# B&R Automation Studio project AS (part 3)

### paiHmiDropdwMenuRT.typ - Global data types
```iecst
(********************************************************************
 * COPYRIGHT -- pai
 ********************************************************************
 * Package: HMI
 * File: HMI.typ
 * Author: goran
 * Created: August 28, 2013
 ********************************************************************
 * Data types of package HMI
 ********************************************************************)
(*########################################################################*)
(*HMI object - Dropdown Menu located at the Upper Right side of the screen*)
(*########################################################################*)

TYPE
	paiHmiDropdwMenuRT_typ : 	STRUCT
		iMenuIndexRT : INT;
		iMenuRTTimeout : REAL; (*Duration after which a dropdown menu is automaticaly hiden if not clicked *)
		oMenuIndexRT : INT; (*Main menu currently selected menu item - RT*)
		oMenuVisible : INT;
		oMenuVisibleItems : ARRAY[0..paiHMI_ENUM_MENU_ITEMS_RT]OF INT; (*1-items is not visible*)
		oMenuDisabledItems : ARRAY[0..paiHMI_ENUM_MENU_ITEMS_RT]OF BOOL; (*1-Item is disabled*)
		iMenuSelectItem : ARRAY[0..paiHMI_ENUM_MENU_ITEMS_RT]OF BOOL; (*an input array to select items from the code; first found 1 will be selected;*)
		oMenuSelectedItems : ARRAY[0..paiHMI_ENUM_MENU_ITEMS_RT]OF BOOL; (*1-Item is currently selected (indexRT)*)
		oMenuPressedItems : ARRAY[0..paiHMI_ENUM_MENU_ITEMS_RT]OF BOOL; (*1-an item that was pressed, single shot*)
		mMenuVisibleOld : INT;
		menuRTHideTimer : TON;
	END_STRUCT;
END_TYPE
```

### paiHmiAlert.h
```c
/********************************************************************
 * COPYRIGHT -- pai
 ********************************************************************
 * Program: hmilogic
 * File: hmiAlert.h
 * Author: goran
 * Created: September 05, 2013
 *******************************************************************/

#include <bur/plctypes.h>
#ifdef _DEFAULT_INCLUDES
#include <AsDefault.h>
#endif
void paiHmiAlertHide(paiHmiAlert_typ* p);
BOOL paiHmiAlertIsActive(paiHmiAlert_typ* p);
void paiHmiAlertShow(paiHmiAlert_typ* p, char* headerText, char* alertText, UDINT alertDuration);
void paiHmiAlertCyclic(paiHmiAlert_typ* p);
```

### paiHmiSystemDateTime.c
```c
/********************************************************************
 * COPYRIGHT -- pai
 ********************************************************************
 * Program: hmilogic
 * File: hmiAlert.c
 * Author: goran
 * Created: September 05, 2013
 *******************************************************************/

#include <bur/plctypes.h>
#ifdef _DEFAULT_INCLUDES
	#include <AsDefault.h>
#endif

void paiHmiSystemDateTimeInit(paiHmiSystemTime_typ* p)
{
}
void paiHmiSystemDateTimeCyclic(paiHmiSystemTime_typ* p)
{
	if(!p->iChangeTimeRequest){
		p->mGetTime.enable = 1;
		p->mGetTime.DT1 = (UDINT)&p->mDateTime;
		DTGetTime(&p->mGetTime);
		p->mDateTime = p->mGetTime.DT1;
		DT_TO_DTStructure(p->mDateTime, (UDINT)&p->oDateTimeActual);
	}else{
		p->iChangeTimeRequest = 0;
		p->mDateTime = DTStructure_TO_DT((UDINT)&p->oDateTimeActual);
		p->mSetTime.enable = 1;
		p->mSetTime.DT1 = p->mDateTime;
		DTSetTime(&p->mSetTime);
	}

}
//eof
```

### paiHmiParamList.h
```c
/********************************************************************
 * COPYRIGHT -- pai
 ********************************************************************
 * Program: hmilogic
 * File: hmiParamList.h
 * Author: goran
 * Created: September 05, 2013
 *******************************************************************/
#include <bur/plctypes.h>
#ifdef _DEFAULT_INCLUDES
#include <AsDefault.h>
#endif
//void hmiParamListTableCyclic(hmiParamListTable_typ* p);
void hmiParamListTableEntryLast(hmiParamListTable_typ* p);
void hmiParamListTableEntryFirst(hmiParamListTable_typ* p, char* pListName);
 void hmiParamListTableAddEntryNext(hmiParamListTable_typ* p, UDINT pValue, char* pName, REAL valDefault, REAL valMin, REAL valMax, int decPlaces, REAL k_factor, REAL n_factor, UINT valueType, char* pDescription);
```

### paiHMI.var
```iecst
(********************************************************************
 * COPYRIGHT -- pai
 ********************************************************************
 * Package: HMI
 * File: HMI.var
 * Author: goran
 * Created: August 28, 2013
 ********************************************************************
 * Variables of package HMI
 ********************************************************************)
VAR
	gPaiHmiMain : paiHmiTemplate_typ; (*HMI logic, page navigation, visibility control, etc.*)
	gPaiHmiMsgScroll : paiHmiMsgScrolling_typ; (*Scrolling Alarm Msg Support*)
	gPaiHmiDialogMsg : paiHmiDialog_typ; (*Scrolling Alarm Msg Support*)
	gPaiHmiAlertMsg : paiHmiAlert_typ; (*Scrolling Alarm Msg Support*)
	gPaiHmiRTMenu : paiHmiDropdwMenuRT_typ;
	gPaiHmiSystemDateTime : paiHmiSystemTime_typ;
	gPaiHmiNetworking : paiHmiSystemNetworking_typ;
END_VAR
VAR RETAIN
	gScrensaverTimeout : INT := 0;
END_VAR
```

### Program Logical/paiComponents/paiTemplate/paiHMI/paiHmi (ANSIC)

- paiHmiSystemDateTime.c (reference to Logical/paiComponents/paiHmi/paiHmiSystemDateTime.c)

### cfgUdpApp.typ - Package data types
```iecst
(********************************************************************
 * COPYRIGHT --
 ********************************************************************
 * Package: UDP
 * File: cfgUdpApp.typ
 * Author: goran
 * Created: October 15, 2014
 ********************************************************************
 * Data types of package UDP
 ********************************************************************)

TYPE
	cfgUdpApp_typ : 	STRUCT
		test1 : UDINT;
		test2 : UDINT;
	END_STRUCT;
END_TYPE
```

- Program Logical/paiComponents/paiUser/paiUser (ANSIC) (no source held here)

### Safety_var.var
```iecst
(*Global PV containing the safety variables.*)
VAR RETAIN
	gSafetyPermInfo : paiSL_Perm_Info_typ;
END_VAR
(*Insert your comment here.*)
VAR
	gSafety : paiSL_typ;
END_VAR
(*Defined constants- change based on specific commissioning configuration*)
VAR
	DEFINE_OFFSET_ERR_START : UDINT := 100000;
END_VAR
VAR CONSTANT
	DEFINE_SAFETY_APP_ID : UINT := 1;
	DEFINE_TIME_MAX_RCTRL_CMD : REAL := 30;
	DEFINE_TIME_ERROR_AUTORESET : REAL := 5;
	DEFINE_TIME_SCANNING_RETRY : REAL := 10;
	DEFINE_TIME_PRINT_HMI_STATUS : REAL := 2;
	DEFINE_SAFELOGIC_ADDRESS : STRING[80] := 'SL1.IF1.ST4.IF1.ST2';
	DEFINE_VERSION : UINT := safeVERSION_R107;
	DEFINE_SAFELOGIC_ID : UINT := 1;
END_VAR
```

### Program Logical/pkgSafety/SafeINIT (IEC)

#### Action_Reset_FBK.st
```iecst
ACTION Action_Reset_FBK:
	gSafety.prv.FBK.RemoteControl.Execute := FALSE;
	gSafety.prv.FBK.DownloadApplication.Execute := FALSE;
	gSafety.prv.FBK.UDID_High.enable := FALSE;
	gSafety.prv.FBK.UDID_Low.enable := FALSE;
END_ACTION
```

### Data object Logical/acp10etxen (Ett)

- acp10etxen.ett (not shown)

- Project.language (not shown)

### Package Logical/HMI - HMI screens 

- Visualisation Logical/HMI/WSVGA (not shown)

### HMImsgScroll.typ - not listed in the package file held
```iecst
(********************************************************************
 * COPYRIGHT -- piedmont
 ********************************************************************
 * Package: HMI
 * File: HMI.typ
 * Author: goran
 * Created: August 28, 2013
 ********************************************************************
 * Data types of package HMI
 ********************************************************************)
(*########################################################################*)
(*HMI object - Scrolling Messages (i.e. alarms)*)
(*########################################################################*)

TYPE
	hmiMsgScrolling_typ : 	STRUCT
		iAdrAlarmArray : UDINT; (*input: address of the alarm array*)
		iAlarmArrayLen : UDINT; (*input: number of alarms in the alarm array*)
		iMsgTimeXms : UDINT; (*input: duration of the message display (if more than one message/alarm active)*)
		oMsgID : UINT; (*output: message ID of the active alarm / message*)
		oMsgVisible : UINT; (*output: visibilty control DP for the VC text message*)
		state : UINT; (*Status for common dialog layer*)
		tmr1 : TON; (*Dialog control timer*)
	END_STRUCT;
END_TYPE
```

### Program Logical/HMI/hmilogic

#### hmiAlert.c
```c
/********************************************************************
 * COPYRIGHT -- piedmont
 ********************************************************************
 * Program: hmilogic
 * File: hmiAlert.c
 * Author: goran
 * Created: September 05, 2013
 *******************************************************************/

#include <bur/plctypes.h>
#ifdef _DEFAULT_INCLUDES
	#include <AsDefault.h>
#endif

/**
Bit manipulaiton utility functions.
 */
//#include <../../bglib/bgBitUtilities.h>

/**
String manipulaiton utility functions.
 */
//#include <../../bglib/bgsprintf.h>
//#include <../../bglib/bgstring.h>

/**
 Timer control utility functions.
 */
//#include <../../bglib/bgTimer1ms.h>

//Control on/off a variable that control the visibility of the alarm alert display
void hmiAlertHide(hmiAlert_typ* p)
{
	//control visibility of the layer > make it invisible
	bgBitSetUINT(&p->status, 0, 1);
}

// Is alert message active (visible)?
BOOL hmiAlertIsActive(hmiAlert_typ* p)
{
	if(bgTimerIsTimeOut(&p->tmr1))
		return 0;
	else
		return 1;
}

// Show the alert with a specified text and for a selected amount of time
void hmiAlertShow(hmiAlert_typ* p, char* alertText, UDINT alertDuration)
{
	//control visibility of the layer > make it visible
	bgBitSetUINT(&p->status, 0, 0);
	bgStrCpyN(p->message, alertText, sizeof(p->message));
	bgTimerStart(&p->tmr1, alertDuration);
}

// Cyclic operation of the alert box.
void hmiAlertCyclic(hmiAlert_typ* p)
{
	bgTimerCyclic(&p->tmr1);
	if( !(p->status & 0x1) && bgTimerIsTimeOut(&p->tmr1) ){
		hmiAlertHide(p);
	}
}
//eof
```

#### hmiDialog.c
```c
/********************************************************************
 * COPYRIGHT -- piedmont
 ********************************************************************
 * Program: hmilogic
 * File: hmiDialog.c
 * Author: goran
 * Created: September 05, 2013
 *******************************************************************/

#include <bur/plctypes.h>
#ifdef _DEFAULT_INCLUDES
	#include <AsDefault.h>
#endif

/*
###############################################################################
Simple dialog support w. OK and Cancle response
###############################################################################
*/

/**
Find if HMI dialog is active (visible) or not
\param p prt to hmiDialog_typ structure
\return 0 not active (not visible)
\return 1 active (visible)
*/
BOOL hmiDialogIsActive(hmiDialog_typ* p)
{
	//hide the dialog
	if(p->status & 0x1){
		return 0; //not visible > not active
	}

	return 1; //visible > active
}

/**
Hide HMI dialog (make it not visible)
\param p prt to hmiDialog_typ structure
*/
void hmiDialogHide(hmiDialog_typ* p)
{
	//hide the dialog
	bgBitSetUINT(&p->status, 0, 1);

	//define the message
	strcpy(p->message, "");
}

/**
Hide HMI dialog (make it not visible)
\param p prt to hmiDialog_typ structure
\param msg text message that will be displayed in a dialog
\param timeout_ms time duration to show the dialog. Upon timer expiration, dialog will automatically generate either ok or cancel (configured, see timeoutConfig)
\param resultForOk value returned in case user response is OK (if 0, default is used = 1)
\param resultForCancel value returned in case user response is Cancel ((if 0, default is used = 2)
\param timeoutConfig 0-timeout wil return value for Cancel, 1-timeout will return value for OK
*/
 void hmiDialogShow(hmiDialog_typ* p, char* msg, UINT timeout_ms, UINT resultForOk, UINT resultForCancel, UINT timeoutConfig)
{
	//show the dialog
	bgBitSetUINT(&p->status, 0, 0);

	//define the message
	bgStrCpyN(p->message, msg, sizeof(p->message));

	//start the timer
	bgTimerStart(&p->tmr1, timeout_ms);

	//set the result to 0 (not complete)
	p->result = 0;
	p->btnOk = 0;
	p->btnCancel = 0;

	//configuration of the timeout
	p->timeoutConfig = timeoutConfig;

	p->resultForOk = resultForOk;
	if(!p->resultForOk)
		p->resultForOk = 1;

	p->resultForCancel = resultForCancel;
	if(!p->resultForCancel)
		p->resultForCancel = 2;

}

/**
Hide HMI dialog cyclic routine
\param p prt to hmiDialog_typ structure
*/
UINT hmiDialogCyclic(hmiDialog_typ* p)
{
	//operate timer always
	bgTimerCyclic(&p->tmr1);

	p->tmr1RemainingTimeSec = (p->tmr1.PT - p->tmr1.ET) / 1000;

	//if dialog not visible > nothing to do
	if(p->status)
		return 0;

	if( bgTimerIsTimeOut(&p->tmr1) ){
		//hide the dialog
		hmiDialogHide(p);
		//check how is the timeout configured and generate such result
		if(!p->timeoutConfig){
			p->result = p->resultForCancel;
			return p->resultForCancel; //return cancel
		}
		p->result = p->resultForOk;
		return p->resultForOk;//return OK
	}

	//keep checking if OK or Cancel buttons are pressed
	if( p->btnOk || p->btnCancel ){

		//hide the dialog
		hmiDialogHide(p);

		//return user's selection:
		if(p->btnOk){
			p->result = p->resultForOk;
		}else
		if(p->btnCancel){
			p->result = p->resultForCancel;
		}

		p->btnOk = 0;
		p->btnCancel = 0;

		return p->result; //return user's selection
	}
	return 0; //no button pressed
}
//EOF
```

### ParStructs.typ
```iecst
(*Insert your comment here.*)

TYPE
	Global_Rec_Cfg_typ : 	STRUCT
		Rec : Global_Rec_typ;
		Cfg : Global_Cfg_typ;
	END_STRUCT;
END_TYPE

(*Insert your comment here.*)

TYPE
	Global_RecCfg_Public_In_typ : 	STRUCT
		Copy_save_to_active : USINT;
		Copy_active_to_save : USINT;
		FileName : STRING[255];
	END_STRUCT;
	Global_RecCfg_Public_Out_typ : 	STRUCT
		save_differs_from_active : USINT;
	END_STRUCT;
	Global_Rec_Cfg_Info_typ : 	STRUCT
		O : Global_RecCfg_Public_Out_typ;
		I : Global_RecCfg_Public_In_typ;
	END_STRUCT;
	Global_Rec_Cfg_IO_typ : 	STRUCT
		Rec : Global_Rec_Cfg_Info_typ;
		Cfg : Global_Rec_Cfg_Info_typ;
	END_STRUCT;
END_TYPE

(*Insert your comment here.*)

TYPE
	Global_Par_typ : 	STRUCT
		save : Global_Rec_Cfg_typ;
		active : Global_Rec_Cfg_typ;
		IO : Global_Rec_Cfg_IO_typ;
	END_STRUCT;
END_TYPE
```

### RecCfg.var
```iecst
VAR CONSTANT
	DEFINE_CONSTANT_MAGIC_PREFIX : UDINT := 16#12345678;
	DEFINE_CONSTANT_MAGIC_SUFFIX : UDINT := 16#87654321;
END_VAR
(*Insert your comment here.*)
VAR CONSTANT
	MAX_IDX_TOTAL_RECIPES : UINT := 100;
END_VAR
(*Insert your comment here.*)
VAR RETAIN
	gConfigName : STRING[255];
	gRecipeName : STRING[255];
END_VAR
(*Insert your comment here.*)
VAR RETAIN
	gRecCfg : Global_Par_typ;
END_VAR
```

### Program Logical/pkgRecCfg/Recipe_Handling (IEC)

#### Init.st - Init code
```iecst
PROGRAM _INIT
	IF gRecCfg.active.Cfg.MagicPrefix <> DEFINE_CONSTANT_MAGIC_PREFIX OR gRecCfg.save.Cfg.MagicPrefix <> DEFINE_CONSTANT_MAGIC_PREFIX
		OR gRecCfg.active.Cfg.MagicSuffix <> DEFINE_CONSTANT_MAGIC_SUFFIX OR gRecCfg.save.Cfg.MagicSuffix <> DEFINE_CONSTANT_MAGIC_SUFFIX THEN

		brsmemset(ADR(gRecCfg.save.Cfg), 0, SIZEOF(Global_Cfg_typ));
		brsmemset(ADR(gRecCfg.active.Cfg), 0, SIZEOF(Global_Cfg_typ));

		gRecCfg.active.Cfg.MagicPrefix := DEFINE_CONSTANT_MAGIC_PREFIX;
		gRecCfg.save.Cfg.MagicPrefix:= DEFINE_CONSTANT_MAGIC_PREFIX;

		gRecCfg.active.Cfg.MagicSuffix := DEFINE_CONSTANT_MAGIC_SUFFIX;
		gRecCfg.save.Cfg.MagicSuffix:= DEFINE_CONSTANT_MAGIC_SUFFIX;
		//
//		brsmemset(ADR(gLinePermData), 0, SIZEOF(Line_Permanent_Variables_typ));
//		brsmemset(ADR(gStatistics), 0, SIZEOF(Global_Statistics_typ));
//		brsmemset(ADR(Axis_Line_Par), 0, SIZEOF(MpAxisBasicParType));
//		brsmemset(ADR(Axis_Blank_Par), 0, SIZEOF(MpAxisBasicParType));
//		brsmemset(ADR(Axis_Coupling_Master_Line_Par), 0, SIZEOF(MpAxisCouplingParType));
//
//		Set_Default_Config_Values(pCfg := ADR(gRecCfg.defaultvals.Cfg), MachineType := gMachineType);
//		Set_Default_Config_Values(pCfg := ADR(gRecCfg.save.Cfg), MachineType := gMachineType);
//		Set_Default_Config_Values(pCfg := ADR(gRecCfg.active.Cfg), MachineType := gMachineType);
//
//		gRecipeName := 'No Config';
//
//		gAlarms.RecCfg.Default_Cfg_Set := TRUE;

//		SYSreset(1, 1);
	END_IF;

	IF gRecCfg.active.Rec.MagicPrefix <> DEFINE_CONSTANT_MAGIC_PREFIX OR gRecCfg.save.Rec.MagicPrefix <> DEFINE_CONSTANT_MAGIC_PREFIX
		OR gRecCfg.active.Rec.MagicSuffix <> DEFINE_CONSTANT_MAGIC_SUFFIX OR gRecCfg.save.Rec.MagicSuffix <> DEFINE_CONSTANT_MAGIC_SUFFIX THEN

		brsmemset(ADR(gRecCfg.save.Rec), 0, SIZEOF(Global_Rec_typ));
		brsmemset(ADR(gRecCfg.active.Rec), 0, SIZEOF(Global_Rec_typ));

		gRecCfg.active.Rec.MagicPrefix := DEFINE_CONSTANT_MAGIC_PREFIX;
		gRecCfg.save.Rec.MagicPrefix:= DEFINE_CONSTANT_MAGIC_PREFIX;

		gRecCfg.active.Rec.MagicSuffix := DEFINE_CONSTANT_MAGIC_SUFFIX;
		gRecCfg.save.Rec.MagicSuffix:= DEFINE_CONSTANT_MAGIC_SUFFIX;
		//
//		brsmemset(ADR(gLinePermData), 0, SIZEOF(Line_Permanent_Variables_typ));
//		brsmemset(ADR(gStatistics), 0, SIZEOF(Global_Statistics_typ));
//		brsmemset(ADR(Axis_Line_Par), 0, SIZEOF(MpAxisBasicParType));
//		brsmemset(ADR(Axis_Blank_Par), 0, SIZEOF(MpAxisBasicParType));
//		brsmemset(ADR(Axis_Coupling_Master_Line_Par), 0, SIZEOF(MpAxisCouplingParType));
//
//		Set_Default_Recipe_Values(pRec := ADR(gRecCfg.defaultvals.Rec), MachineType := gMachineType);
//		Set_Default_Recipe_Values(pRec := ADR(gRecCfg.save.Rec), MachineType := gMachineType);
//		Set_Default_Recipe_Values(pRec := ADR(gRecCfg.active.Rec), MachineType := gMachineType);
//
//		gRecipeName := 'No Recipe';
//
//		gAlarms.RecCfg.Default_Rec_Set := TRUE;
//		SYSreset(1, 1);
	END_IF;

	gRecCfg.IO.Rec.I.FileName := 'rec1';
	gRecCfg.IO.Cfg.I.FileName := 'cfg1';

	Recipe_CSV_Control.MpLink := ADR(Recipe_CSV_MpLink);
	Recipe_CSV_Control.Enable := TRUE;
	Recipe_CSV_Control.DeviceName := ADR('Recipe');
	Recipe_CSV_Control.FileName := ADR(gRecCfg.IO.Rec.I.FileName);
	Recipe_CSV_Control.Category := ADR('Recipe');
	Recipe_CSV_Control.Header := ADR(Recipe_CSV_Header);

	Config_CSV_Control.MpLink := ADR(Config_CSV_MpLink);
	Config_CSV_Control.Enable := TRUE;
	Config_CSV_Control.DeviceName := ADR('Config');
	Config_CSV_Control.FileName := ADR(gRecCfg.IO.Cfg.I.FileName);
	Config_CSV_Control.Category := ADR('Config');
	Config_CSV_Control.Header := ADR(Config_CSV_Header);

	Recipe_CSV_RegPar.MpLink := ADR(Recipe_CSV_MpLink);
	Recipe_CSV_RegPar.Enable := TRUE;
	Recipe_CSV_RegPar.PVName := ADR('gRecCfg.save.Rec');
	Recipe_CSV_RegPar.Category := ADR('Recipe');

	Config_CSV_RegPar.MpLink := ADR(Config_CSV_MpLink);
	Config_CSV_RegPar.Enable := TRUE;
	Config_CSV_RegPar.PVName := ADR('gRecCfg.save.Cfg');
	Config_CSV_RegPar.Category := ADR('Config');

	Recipe_CSV_UI.MpLink := ADR(Recipe_CSV_MpLink);
	Recipe_CSV_UI.Enable := TRUE;
	Recipe_CSV_UI.UIConnect := ADR(gRecipe_CSV_UIConnect);

	Config_CSV_UI.MpLink := ADR(Config_CSV_MpLink);
	Config_CSV_UI.Enable := TRUE;
	Config_CSV_UI.UIConnect := ADR(gConfig_CSV_UIConnect);

	Recipe_CSV_UI.UISetup.RecipeListSize := 20;
	Recipe_CSV_UI.UISetup.RecipeListScrollWindow := 1;
	Recipe_CSV_UI.UISetup.Confirmation.RecipeCreate := TRUE;
	Recipe_CSV_UI.UISetup.Confirmation.RecipeLoad := TRUE;
	Recipe_CSV_UI.UISetup.Confirmation.RecipeSave := TRUE;
	Recipe_CSV_UI.UISetup.Confirmation.RecipeDelete := TRUE;

	Config_CSV_UI.UISetup.RecipeListSize := 20;
	Config_CSV_UI.UISetup.RecipeListScrollWindow := 1;
	Config_CSV_UI.UISetup.Confirmation.RecipeCreate := TRUE;
	Config_CSV_UI.UISetup.Confirmation.RecipeLoad := TRUE;
	Config_CSV_UI.UISetup.Confirmation.RecipeSave := TRUE;
	Config_CSV_UI.UISetup.Confirmation.RecipeDelete := TRUE;

	pRecCfgUIConnect ACCESS ADR(gRecipe_CSV_UIConnect);
	pCmd ACCESS ADR(loc.Rec.HMI);

	gRecipe_CSV_UIConnect.New.FileName := 'Rec_Name';
	gConfig_CSV_UIConnect.New.FileName := 'Cfg_Name';

	Recipe_CSV_Control;
	Recipe_CSV_RegPar;
	Recipe_CSV_UI;

	Config_CSV_Control;
	Config_CSV_RegPar;
	Config_CSV_UI;

END_PROGRAM
```

### Alarm.var
```iecst
VAR
	AlarmX_HistoryUI : MpAlarmXHistoryUI;
	AlarmX_History_UIConnect : MpAlarmXHistoryUIConnectType;
	AlarmX_ListUI : MpAlarmXListUI;
	AlarmX_ListUIConnect : MpAlarmXListUIConnectType;
	AlarmX_History : MpAlarmXHistory;
	AlarmX_Control : MpAlarmXCore;
END_VAR
(*Insert your comment here.*)
VAR
	Com_Logger_UI : MpComLoggerUI := (0);
	Com_Logger_UIConnect : MpComLoggerUIConnectType := (0);
END_VAR
```

### Program Logical/pkgAlert/AlarmX (IEC)

#### Types.typ
```iecst
TYPE
	MachineAlarm_typ : 	STRUCT
		str : {REDUND_UNREPLICABLE} STRING[80];
		active : {REDUND_UNREPLICABLE} BOOL;
	END_STRUCT;
	MachineReaction_typ : 	STRUCT
		str : {REDUND_UNREPLICABLE} STRING[80];
		active : {REDUND_UNREPLICABLE} BOOL;
	END_STRUCT;
	AlarmX_Local_TmpVar_typ : 	STRUCT
		val_float : {REDUND_UNREPLICABLE} REAL;
		ExampleAlarm : {REDUND_UNREPLICABLE} MachineAlarm_typ;
		ExampleReaction : {REDUND_UNREPLICABLE} MachineReaction_typ;
	END_STRUCT;
END_TYPE
```

### UserXVar.var
```iecst
VAR
	UserX_ManagerUI : MpUserXManagerUI;
	UserX_LoginUI : MpUserXLoginUI;
	UserX_Login : MpUserXLogin;
END_VAR
```

### Program Logical/pkgData/DataTask (IEC)

#### LocalFunctions.fun
```iecst
FUNCTION Register_Log_PV : BOOL (* *) (*$GROUP=User,$CAT=User,$GROUPICON=User.png,$CATICON=User.png*)
	VAR_INPUT
		pDesc : REFERENCE TO STRING[80]; (*pRegParBlock : REFERENCE TO MpDataRegPar;*)
		pPVName : REFERENCE TO STRING[80];
		pIterator : REFERENCE TO DINT;
		pMpLink : REFERENCE TO MpComIdentType;
	END_VAR
END_FUNCTION
```

#### Register_Log_PV.st
```iecst
FUNCTION Register_Log_PV

//	pRegParBlock.MpLink := ADR(pMpLink);
//	pRegParBlock.Enable := TRUE;
//	pRegParBlock.PVName := ADR(pPVName);
//	pRegParBlock.Description := ADR(pDesc);
//	pRegParBlock();

	pIterator := pIterator + 1;
	RETURN;
END_FUNCTION
```

### Program Logical/pkgData/File_Handling (IEC)

#### Init.st - Init code
```iecst
PROGRAM _INIT
	File_Manager_Control.MpLink := ADR(File_Manager_MpLink);
	File_Manager_Control.Enable := TRUE;
	File_Manager_Control.UIConnect := ADR(File_Manager_UIConnect);

	File_Manager_UIConnect.DeviceList.DeviceNames[0] := 'ROOT';
	File_Manager_UIConnect.DeviceList.DeviceNames[1] := 'Config';
	File_Manager_UIConnect.DeviceList.DeviceNames[2] := 'Recipe';
	File_Manager_UIConnect.DeviceList.DeviceNames[3] := 'Data_Log';
	File_Manager_UIConnect.DeviceList.DeviceNames[4] := 'USB1';
	File_Manager_UIConnect.DeviceList.DeviceNames[5] := 'USB2';

	File_Manager_Control.UISetup.FileListSize := 8;
	File_Manager_Control.UISetup.FileListScrollWindow := 5;

	File_Manager_Control;

END_PROGRAM
```

### Library Logical/pkgPVListView/paiPVTable (ANSIC)
Depends on: standard, sys_lib, wbrLogSvc, ArTextSys, bglibasWBR, jgLibC, Acp10par

#### Languages.typ
```iecst
TYPE
	Language_Enums :
		(
		LANGUAGE_ENGLISH := 0,
		LANGUAGE_SWEDISH := 1,
		LANGUAGE_PORTUGESE := 2,
		LANGUAGE_GERMAN := 3,
		LANGUAGE_FRENCH := 4,
		LANGUAGE_SPANISH := 5
		);
	Enum_PV_types :
		(
		PV_REAL,
		PV_UDINT
		);
END_TYPE
```

### Program Logical/pkgPVListView/HMITableManager (IEC)

#### Types.typ
```iecst
TYPE
	hmiTableRecCfgTrigger_typ : 	STRUCT
		Dispense : BOOL := FALSE;
		Inspect : BOOL := FALSE;
	END_STRUCT;
	hmiTableTrigger_typ : 	STRUCT
		Rec : hmiTableRecCfgTrigger_typ;
		Cfg : hmiTableRecCfgTrigger_typ;
	END_STRUCT;
	hmiTableLoad_typ : 	STRUCT
		Trigger : BOOL;
	END_STRUCT;
	hmiTables_typ : 	STRUCT
		Trigger : hmiTableTrigger_typ;
		Load : hmiTableLoad_typ;
	END_STRUCT;
	HMITableControlLocal_typ : 	STRUCT
		tables : hmiTables_typ;
	END_STRUCT;
END_TYPE
```

#### Main.st
```iecst
PROGRAM _INIT
	Init_Logbook.Enable := TRUE;
	Init_Logbook.Name := 'usr_table';
	Init_Logbook();

END_PROGRAM

//TODO: Load param array with %s, replace with index.
//TODO: More scrutiny to ensure tables were done correctly

PROGRAM _CYCLIC
	svnRevision;

//	IF loc.tables.Trigger.Rec.Dispense THEN
//		loc.tables.Trigger.Rec.Dispense := FALSE;
//		ActivateHMITable(gRecCfg.active.Cfg.HMI.MachineLang, pHMITable := ADR(gHmiParamTable), pTableValues := ADR(loadHMITable[TABLE_REC_DISPENSE].hmiStruct));
//	END_IF;
//
//	IF loc.tables.Trigger.Rec.Inspect THEN
//		loc.tables.Trigger.Rec.Inspect := FALSE;
//		ActivateHMITable(gRecCfg.active.Cfg.HMI.MachineLang, pHMITable := ADR(gHmiParamTable), pTableValues := ADR(loadHMITable[TABLE_REC_INSPECT].hmiStruct));
//	END_IF;
//
//	IF loc.tables.Trigger.Rec.Eject THEN
//		loc.tables.Trigger.Rec.Eject := FALSE;
//		ActivateHMITable(gRecCfg.active.Cfg.HMI.MachineLang, pHMITable := ADR(gHmiParamTable), pTableValues := ADR(loadHMITable[TABLE_REC_EJECT].hmiStruct));
//	END_IF;
//
//	IF loc.tables.Trigger.Rec.Motor THEN
//		loc.tables.Trigger.Rec.Motor := FALSE;
//		ActivateHMITable(gRecCfg.active.Cfg.HMI.MachineLang, pHMITable := ADR(gHmiParamTable), pTableValues := ADR(loadHMITable[TABLE_REC_MOTOR].hmiStruct));
//	END_IF;
//
//	IF loc.tables.Trigger.Rec.Process THEN
//		loc.tables.Trigger.Rec.Process := FALSE;
//		ActivateHMITable(gRecCfg.active.Cfg.HMI.MachineLang, pHMITable := ADR(gHmiParamTable), pTableValues := ADR(loadHMITable[TABLE_REC_PROCESS].hmiStruct));
//	END_IF;
//
//	IF loc.tables.Trigger.Rec.Loader THEN
//		loc.tables.Trigger.Rec.Loader := FALSE;
//		ActivateHMITable(gRecCfg.active.Cfg.HMI.MachineLang, pHMITable := ADR(gHmiParamTable), pTableValues := ADR(loadHMITable[TABLE_REC_LOADER].hmiStruct));
//	END_IF;
//
//	IF loc.tables.Trigger.Cfg.Dispense THEN
//		loc.tables.Trigger.Cfg.Dispense := FALSE;
//		ActivateHMITable(gRecCfg.active.Cfg.HMI.MachineLang, pHMITable := ADR(gHmiParamTable), pTableValues := ADR(loadHMITable[TABLE_CFG_DISPENSE].hmiStruct));
//	END_IF;
//
//	IF loc.tables.Trigger.Cfg.Inspect THEN
//		loc.tables.Trigger.Cfg.Inspect := FALSE;
//		ActivateHMITable(gRecCfg.active.Cfg.HMI.MachineLang, pHMITable := ADR(gHmiParamTable), pTableValues := ADR(loadHMITable[TABLE_CFG_INSPECT].hmiStruct));
//	END_IF;
//
//	IF loc.tables.Trigger.Cfg.Eject THEN
//		loc.tables.Trigger.Cfg.Eject := FALSE;
//		ActivateHMITable(gRecCfg.active.Cfg.HMI.MachineLang, pHMITable := ADR(gHmiParamTable), pTableValues := ADR(loadHMITable[TABLE_CFG_EJECT].hmiStruct));
//	END_IF;
//
//	IF loc.tables.Trigger.Cfg.Motor THEN
//		loc.tables.Trigger.Cfg.Motor := FALSE;
//		ActivateHMITable(gRecCfg.active.Cfg.HMI.MachineLang, pHMITable := ADR(gHmiParamTable), pTableValues := ADR(loadHMITable[TABLE_CFG_MOTOR].hmiStruct));
//	END_IF;
//
//	IF loc.tables.Trigger.Cfg.Process THEN
//		loc.tables.Trigger.Cfg.Process := FALSE;
//		ActivateHMITable(gRecCfg.active.Cfg.HMI.MachineLang, pHMITable := ADR(gHmiParamTable), pTableValues := ADR(loadHMITable[TABLE_CFG_PROCESS].hmiStruct));
//	END_IF;
//
//	IF loc.tables.Trigger.Cfg.Loader THEN
//		loc.tables.Trigger.Cfg.Loader := FALSE;
//		ActivateHMITable(gRecCfg.active.Cfg.HMI.MachineLang, pHMITable := ADR(gHmiParamTable), pTableValues := ADR(loadHMITable[TABLE_CFG_LOADER].hmiStruct));
//	END_IF;
//
//	IF loc.tables.Trigger.Cfg.Admin THEN
//		loc.tables.Trigger.Cfg.Admin := FALSE;
//		ActivateHMITable(gRecCfg.active.Cfg.HMI.MachineLang, pHMITable := ADR(gHmiParamTable), pTableValues := ADR(loadHMITable[TABLE_CFG_ADMIN].hmiStruct));
//	END_IF;
//
//	IF loc.tables.Load.Trigger THEN
//		SYSreset(1,1);
//	END_IF;
//
//	hmiParamListTableCyclic(ADR(gHmiParamTable));

END_PROGRAM

PROGRAM _EXIT
	(* Insert code here *)

END_PROGRAM
```

### Audit_Global.var
```iecst
VAR
	Audit_Control : MpAuditTrail := (0);
	Audit_Config : MpAuditTrailConfig := (0);
	Audit_Config_Struct : MpAuditTrailConfigType := (0);
	Audit_UI : MpAuditTrailUI := (0);
	Audit_UIConnect : MpAuditTrailUIConnectType := (0);
	Audit_VC4_Event : MpAuditVC4Event := (0);
END_VAR
```

### EnMon_Global.var
```iecst
VAR
	Energy_Control : MpEnergyCore;
	Energy_UI : MpEnergyCoreUI := (UISetup:=(ModuleListSize:=6));
	Energy_UIConnect : MpEnergyCoreUIConnectType;
END_VAR
```

### Program Logical/pkgEnMon/EnMon (IEC)

#### Main.st
```iecst
PROGRAM _INIT
	Energy_Control.MpLink := ADR(Energy_MpLink);
	Energy_Control.Enable := TRUE;
	Energy_Control.DeviceName := ADR('Energy');
	Energy_Control();
	Energy_UI.MpLink := ADR(Energy_MpLink);
	Energy_UI.Enable := TRUE;
	Energy_UI.UISetup.ModuleListSize := 5;
	Energy_UI.UISetup.ModuleScrollWindow := 10;
	Energy_UI.UIConnect := ADR(Energy_UIConnect);
	Energy_UI();
	Energy_UIConnect;
END_PROGRAM

PROGRAM _CYCLIC
	Energy_Control();
	Energy_UI();
	Energy_UIConnect;
END_PROGRAM

PROGRAM _EXIT

END_PROGRAM
```

### Variables.var
```iecst
VAR
	PackML_Basic_UIConnect : MpPackMLBasicUIConnectType;
	PackML_Statistics_UIConnect : MpPackMLStatisticsUIConnectType;
END_VAR
```

### MpView_Aux_Global.var
```iecst
VAR
	gVis : HTMLVis_typ;
END_VAR
```

### Program Logical/pkgMpViewAux/VisCtrl

#### Main.st
```iecst
PROGRAM _INIT

END_PROGRAM

PROGRAM _CYCLIC
	clientSlots;
	usint_tmp;
	gVis;

	gVis.Alert.numAlarms := AlarmX_Control.ActiveAlarms;
	gVis.Alert.numWarnings := AlarmX_Control.PendingAlarms;
	gVis.Alert.idxImage := BOOL_TO_DINT(AlarmX_Control.ActiveAlarms > 0)*2;

	CASE gVis.Motion.indexAxis OF
		0:
			pAxisControl ACCESS ADR(gDelta.jointAxes[0].Control);
			pAxisPar ACCESS ADR(gRecCfg.active.Cfg.Delta.Axes.Joint[0].Par);
		1:
			pAxisControl ACCESS ADR(gDelta.jointAxes[1].Control);
			pAxisPar ACCESS ADR(gRecCfg.active.Cfg.Delta.Axes.Joint[1].Par);
		2:
			pAxisControl ACCESS ADR(gDelta.jointAxes[2].Control);
			pAxisPar ACCESS ADR(gRecCfg.active.Cfg.Delta.Axes.Joint[2].Par);
		3:
			pAxisControl ACCESS ADR(gDelta.jointAxes[3].Control);
			pAxisPar ACCESS ADR(gRecCfg.active.Cfg.Delta.Axes.Joint[3].Par);
		4:
			pAxisControl ACCESS ADR(gDelta.pathAxes[0].Control);
			pAxisPar ACCESS ADR(gRecCfg.active.Cfg.Delta.Axes.Path[0].Par);
		5:
			pAxisControl ACCESS ADR(gDelta.pathAxes[1].Control);
			pAxisPar ACCESS ADR(gRecCfg.active.Cfg.Delta.Axes.Path[1].Par);
		6:
			pAxisControl ACCESS ADR(gDelta.pathAxes[2].Control);
			pAxisPar ACCESS ADR(gRecCfg.active.Cfg.Delta.Axes.Path[2].Par);
		7:
			pAxisControl ACCESS ADR(gDelta.pathAxes[3].Control);
			pAxisPar ACCESS ADR(gRecCfg.active.Cfg.Delta.Axes.Path[3].Par);
	END_CASE;

END_PROGRAM

PROGRAM _EXIT
	(* Insert code here *)

END_PROGRAM
```

- Visualisation Logical/mappView (not shown)

### Data object Logical/GmcIpConfig/gmcipsys (Cnc)

#### gmcipsys.cnc
```
LANGS (defaultLangId=1, defaultDataLangId=3)
  CMDQUEUE (BufferSize=15)
  MEM (ReserveMB=5, LimitPercent=80%)
  EXEC (InstrBurstBG=200, CycleBurstBG=0, Stack=16384, MinorStack=2048, EStack=1024)
  LOAD (ReadLineBurstMax=100, ReadLineBurstMin=20, ParseLineBurstMax=10, ParseLineBurstMin=2, RuntimeIOBlocking=No)
  DISABLE_MSG = 15238 
    15336 
    15337 
    15666 
    15784 
    15864 
    15740
  LANG (langId=1, langName=B&R GCode, langModule=ailgcode)
    LANGCONFIG gmciplbr
    LANGCONFIG gmcipcbr
    LANGCONFIG gmcipubr
    FILEEXT .cnc
    FILEEXT .prg
    MAINSEARCHPATH $ (FileDevice=CNC_PrgDir)
    MAINSEARCHPATH $ (DataObject=Yes)
    INCLUDEPATH $ (FileDevice=CNC_PrgDir)
    INCLUDEPATH $ (DataObject=Yes)
  LANG (langId=2, langName=Alternative Language 1 GCode, langModule=ailgcode)
    LANGCONFIG gmciplsm
    LANGCONFIG gmcipcbr
    LANGCONFIG gmcipcsm
    LANGCONFIG gmcipusm
    FILEPREFIX = _N_
    FILEEXT = .MPF
    FILEEXT = _MPF
    FILEEXT = .SPF
    FILEEXT = _SPF
    MAINSEARCHPATH = \$ (FileDevice=CNC_PrgDir)
    MAINSEARCHPATH = \_N_MPF_DIR\$ (FileDevice=CNC_PrgDir)
    MAINSEARCHPATH = \_N_SPF_DIR\$ (FileDevice=CNC_PrgDir)
    MAINSEARCHPATH = $ (DataObject=1)
    INCLUDEPATH = \$ (FileDevice=CNC_PrgDir)
    INCLUDEPATH = \_N_SPF_DIR\$ (FileDevice=CNC_PrgDir)
    INCLUDEPATH = \_N_MPF_DIR\$ (FileDevice=CNC_PrgDir)
    INCLUDEPATH = $ (DataObject=1)
  LANG (langId=3, langName=IEC-ST, langModule=ailgcode)
    LANGCONFIG gmcipiec
    LANGCONFIG gmcipmx (RequireFnIgnore=MXConvertOrient)
    LANGCONFIG gmcipui (IfNotExist=Warn)
    FILEEXT .typ (DeclScope=IP_GLOBAL)
    FILEEXT .var (DeclScope=IP_GLOBAL)
    FILEEXT .fun (DeclScope=IP_GLOBAL)
    FILEEXT .iec (DeclScope=IP_LOCAL)
    FILEEXT .st (DeclScope=IP_LOCAL)
    FILEEXT _iec (DeclScope=IP_LOCAL)
    MAINSEARCHPATH = \$ (FileDevice=IEC_PrgDir)
    MAINSEARCHPATH = \$ (FileDevice=CNC_PrgDir)
    MAINSEARCHPATH \TYP\$ (FileDevice=CNC_PrgDir, DataObject=No)
    INCLUDEPATH = \$ (FileDevice=IEC_PrgDir)
    INCLUDEPATH = \$ (FileDevice=CNC_PrgDir)
    INCLUDEPATH \TYP\$ (FileDevice=CNC_PrgDir, DataObject=No)
  XML_INCLUDE gmcipus (IfNotExist=Warn)
```

### Data object Logical/GmcIpConfig/gmcipcbr (Cnc, version 3.14.3)

- gmcipcbr.cnc (not shown)

### Data object Logical/GmcIpConfig/gmciplsm (Cnc, version 3.14.3)

#### gmciplsm.cnc
```
Root (LangModule=ailgcode, Version=1.0)
  PrimTypes (CaseSensitive=No)
    REAL (BRType=LREAL)
    INT (BRType=DINT)
    CHAR (BRType=USINT)
    BOOL (BRType=BOOL)
    STRING (BRType=STRING)
    AXIS (BRType=AXIS)
    BR_LREAL (BRType=LREAL)
    BR_REAL (BRType=REAL)
    BR_UDINT (BRType=UDINT)
    BR_DINT (BRType=DINT)
    BR_UINT (BRType=UINT)
    BR_INT (BRType=INT)
    BR_USINT (BRType=USINT)
    BR_SINT (BRType=SINT)
    BR_BOOL (BRType=BOOL)
    BR_TIME (BRType=TIME)
    BR_DATE_AND_TIME (BRType=DATE_AND_TIME)
  Preprocess:
    PP_RULE_NCK (Search=NCK , Replace=nc_global )
    PP_RULE_CHAN (Search=CHAN , Replace=ip_global )
    PP_RULE_FRAME_I (Search=$FRAME_I, Replace=(1,0,0,0,1,0,0,0,1,0,0,0))
    PP_RULE_FRAME_DEF (IsPattern=Yes, Search=FRAME:[^\w\d], Replace=REAL[12])
  BuiltInProcs:
    cancel = beginpathsynch
        StopCyclicGroups(:${*}:);
      endpathsynch (MinArgs=1, MaxArgs=*)
    RET = #next_motion.Command = MPCMD_SET_M_FCT;
      #next_motion.Data.I4_value = 17;
      PushPacket(::);
      ReturnTo(:${*}:); (MinArgs=0, MaxArgs=4, Eval=Early, Inline=Yes)
  BuiltInFns:
    ABS = Abs(:$[1]:) (NumArgs=1, Inline=Yes)
    SIN = Sin(:$[1]:) (NumArgs=1, Inline=Yes)
    COS = Cos(:$[1]:) (NumArgs=1, Inline=Yes)
    TAN = Tan(:$[1]:) (NumArgs=1, Inline=Yes)
    ASIN = ASin(:$[1]:) (NumArgs=1, Inline=Yes)
    ACOS = ACos(:$[1]:) (NumArgs=1, Inline=Yes)
    ATAN = ATan(:$[1]:) (NumArgs=1, Inline=Yes)
    ATAN2 = ATan2(:$[1],$[2]:) (NumArgs=2, Inline=Yes)
    SQRT = Sqrt(:$[1]:) (NumArgs=1, Inline=Yes)
    POT = (($[1])*($[1])) (NumArgs=1, Inline=Yes)
    TRUNC = Fix(:$[1]:) (NumArgs=1, Inline=Yes)
    ROUND = Round(:$[1]:) (NumArgs=1, Inline=Yes)
    LN = Ln(:$[1]:) (NumArgs=1, Inline=Yes)
    EXP = Exp(:$[1]:) (NumArgs=1, Inline=Yes)
    MINVAL = MinVal(:$[1], $[2]:) (NumArgs=2, Inline=Yes)
    MAXVAL = MaxVal(:$[1], $[2]:) (NumArgs=2, Inline=Yes)
    BOUND = Bounds(:$[1], $[2], $[3]:) (NumArgs=3, Inline=Yes)
    TO_BOOL = ToBool(:$[1]:) (NumArgs=1, Inline=Yes)
    TO_INT = ToInt(:$[1]:) (NumArgs=1, Inline=Yes)
    TO_CHAR = ToChar(:$[1]:) (NumArgs=1, Inline=Yes)
    TO_REAL = ToLReal(:$[1]:) (NumArgs=1, Inline=Yes)
    TO_FLOAT = ToFloat(:$[1]:) (NumArgs=1, Inline=Yes)
    DEFINED = Defined(:$[1]:) (NumArgs=1, Inline=Yes)
    TIME_MS = TimeMs(::) (NumArgs=0)
    SET = ${*} (MinArgs=0, MaxArgs=*, Inline=Yes)
    REP = ArrayRep(:${*}:) (MinArgs=1, MaxArgs=2, Inline=Yes)
    ADR = Adr(:\$[1]:) (NumArgs=1, Inline=Yes)
    SIZEOF = Sizeof(:\$[1]:) (NumArgs=1, Inline=Yes)
    NUM_LOADED_FILES = NumLoadedFiles(::) (NumArgs=0)
    NUM_LOADED_PROG_FILES = NumLoadedProgFiles(::) (NumArgs=0)
    MEM_SIZE_IP_ALL = MemSizeIpInstAll(::) (NumArgs=0)
    MEM_SIZE_IP_LIB = MemSizeIpInst(::) (NumArgs=0)
    MEM_SIZE_SHLIB = MemSizeShLib(::) (NumArgs=0)
    MEM_SIZE_FILE = MemSizeFile(:$[1]:) (MinArgs=0, MaxArgs=1)
    MEM_SIZE_IP_STACK_SPACE = MemStackSpace(::) (NumArgs=0)
  AxesSpec:
    AxisRef = $\s*=\s*AC (Mode=3)
    AxisRef = $\s*=\s*IC (Mode=4)
  PVMacros:
    SBLOF (ArrayDims=0, Group=500)
      CALL = #call->forbid_stepping = 1; (Inline=Yes)
    SBLON (ArrayDims=0, Group=500)
      CALL = #call->forbid_stepping = 0; (Inline=Yes)
    DISPLOF (ArrayDims=0, Group=500)
      CALL = #call->forbid_display = 1; (Inline=Yes)
    DISPLON (ArrayDims=0, Group=500)
      CALL = #call->forbid_display = 0; (Inline=Yes)
    RDISABLE (ArrayDims=0, Group=500)
      CALL = @#job->sa.keep_alive = 1;
        @#thread.sa_keep_alive = 1; (Inline=Yes)
    P_SUBPAR $P_SUBPAR (ArrayDims=1, Group=500)
      GET = return ArgNumIsDefined(:$[1]:);
    P_STACK $P_STACK:
      GET = return UserCallDepth(::);
  FubTemplates:
    StdFubTemplate (IsDefault=Yes, Inline=Yes)
      Arg (ref=FUBINST, DataType=FLOAT)
      Arg (ref=FUBERRLEV, DataType=FLOAT)
      Arg (ref=PATHSYNCH, DataType=FLOAT)
      Arg (ref=BLOCKING, DataType=FLOAT)
  SynchActions:
    SABlocks:
      default (IsDefault=Yes)
        cyclic (Inline=Yes)
          Arg (ref=ACTIONS, DataType=STATEMENTS)
          Arg (ref=ID, DataType=FLOAT, DefaultInt=-1, MinCount=0, MaxCount=1)
      whenever:
        cyclic (Inline=Yes)
          Arg (ref=COND, DataType=FLOAT)
          Arg (ref=ACTIONS, DataType=STATEMENTS)
          Arg (ref=ID, DataType=FLOAT, DefaultInt=-1, MinCount=0, MaxCount=1)
      when:
        cyclic (Inline=Yes)
          Arg (ref=COND, DataType=FLOAT)
          Arg (ref=ACTIONS, DataType=STATEMENTS)
          Arg (ref=ID, DataType=FLOAT, DefaultInt=-1, MinCount=0, MaxCount=1)
      every:
        cyclic (Inline=Yes)
          Arg (ref=COND, DataType=FLOAT)
          Arg (ref=ACTIONS, DataType=STATEMENTS)
          Arg (ref=ID, DataType=FLOAT, DefaultInt=-1, MinCount=0, MaxCount=1)
      from:
        cyclic (Inline=Yes)
          Arg (ref=COND, DataType=FLOAT)
          Arg (ref=ACTIONS, DataType=STATEMENTS)
          Arg (ref=ID, DataType=FLOAT, DefaultInt=-1, MinCount=0, MaxCount=1)
    NonModalActivation:
      Start = @#thread.sa_last_keep_alive = 1;
        ActivateCyclicGroup(:-1:);
      Stop = WaitStopCyclicGroups(:(:-1:):);
  ParserData (NestedComments=Yes, DefaultCaseSensitive=No, CommentsSpanLines=No, SubDeclsLocalToFile=Yes, ProgDeclsLocalToFile=Yes, AllowUnprefixedFileCalls=Yes, AllowUnprefixedSubCalls=Yes, LocalVarScopeForMainProg=No, FileScopeVarsVisibleInSub=Yes, MainPrgReturnAtNextMainPrgHdr=Yes, AllowVarReadBeforeAssign=No, AllowArrayRefWithoutIndex=Yes, AllowNamedFnArgs=Yes, AllowBuiltinFnArgsOutOfSequence=Yes, AllowBuiltInProcCallWithoutBrackets=Yes, AllowBuiltInFnCallWithoutBrackets=No, AllowPLCFnCallWithoutBrackets=No, AllowStructMemberAutoDereference=Yes, AllowVariableAutoDereference=Yes, EnableStringCharacterIndexing=Yes, AllowIgnoredExtraSubArgs=Yes, OnMacroRedefinition=Error, CheckFileTimestampBeforeCalls=Yes)
    TKG_END_OF_LINE = \n (IsPattern=No)
    TKG_LINE_CONTINUE = \ (IsPattern=No, FileXLInvalid=Yes)
    TKG_LINE_BREAK = @@
    TKG_OPEN_COMMENT = ;
    TKG_CLOSE_COMMENT
    TKG_TRUE = TRUE:\W (IsPattern=Yes)
    TKG_FALSE = FALSE:\W (IsPattern=Yes)
    TKG_PAREVAL_MODAL_ID = ID:[\s=] (FileXLInvalid=Yes, IsPattern=Yes)
    TKG_MACRO_DEFINE_GLOBAL = define\s+ip_global:\s (IsPattern=Yes, FollowedBy=TKG_MACRO_NAME)
    TKG_MACRO_DEFINE = define\s+local:\s|define:\s (IsPattern=Yes, FollowedBy=TKG_MACRO_NAME)
    TKG_MACRO_UNDEFINE = undefine:\s (IsPattern=Yes, FollowedBy=TKG_MACRO_NAME)
    TKG_MACRO_AS = as:[\s\n] (IsPattern=Yes, FollowedBy=TKG_MACRO_TEXT)
    TKG_PROG_START = %:[^L] (IsPattern=Yes, CaseSensitive=Yes, FollowedBy=TKG_PROG_NAME)
    TKG_PROG_NAME = [\w\d]+ (IsPattern=Yes, Restricted=Yes)
    TKG_SET_MODAL_SUB = MCALL:\W (FileXLInvalid=Yes, IsPattern=Yes)
    TKG_INDIR_PROG_CALL = CALL:\s (IsPattern=Yes)
    TKG_INDIR_PROG_BLOCK = BLOCK:\s (FileXLInvalid=Yes, IsPattern=Yes)
    TKG_PROC_START = PROC:\s (FileXLInvalid=Yes, IsPattern=Yes, FollowedBy=TKG_PROC_NAME)
    TKG_PROC_NAME = \w[\w\d]+ (IsPattern=Yes, Restricted=Yes)
    TKG_ARG_PASSBYREF = VAR:\s (IsPattern=Yes)
    TKG_SUBPROG_PROTO = INTERN:\s (IsPattern=Yes, FollowedBy=TKG_SUBPROG_NAME)
    TKG_SUBPROG_START = SUB\s|%:L (FileXLInvalid=Yes, IsPattern=Yes, CaseSensitive=Yes, FollowedBy=TKG_SUBPROG_NAME)
    TKG_SUBPROG_NAME = \w[\w\d]+ (IsPattern=Yes, Restricted=Yes)
    TKG_EXTERN = EXTERN:\s (IsPattern=Yes, FollowedBy=TKG_PROG_FILE_NAME)
    TKG_PROG_FILE_NAME = [\^#&@']?[\w\d\./\:]+ (IsPattern=Yes, Restricted=Yes)
    TKG_PV_DECL = def:\s (IsPattern=Yes)
    TKG_PV_UNDECL = ~def:\s (IsPattern=Yes)
    TKG_VAR_RETAIN = retain:\s (IsPattern=Yes)
    TKG_VARSCOPE_IP_LOCAL = local:[\s\n] (IsPattern=Yes)
    TKG_VARSCOPE_IP_GLOBAL = ip_global:[\s\n] (IsPattern=Yes)
    TKG_VARSCOPE_NC_GLOBAL = nc_global:[\s\n] (IsPattern=Yes)
    TKG_VARSCOPE_PLC_GLOBAL = plc_global:[\s\n] (IsPattern=Yes)
    TKG_VARSYNCH_IP = ip_synch:\s (IsPattern=Yes)
    TKG_VARSYNCH_PATH = path_synch:\s (IsPattern=Yes)
    TKG_PAREVAL_DO = do:\s (FileXLInvalid=Yes, IsPattern=Yes)
    TKG_GOTOF = gotof:\s (FileXLInvalid=Yes, IsPattern=Yes, OptFollowedBy=TKG_GOTO_DEST)
    TKG_GOTOB = gotob:\s (FileXLInvalid=Yes, IsPattern=Yes, OptFollowedBy=TKG_GOTO_DEST)
    TKG_GOTO = goto:\s (FileXLInvalid=Yes, IsPattern=Yes, OptFollowedBy=TKG_GOTO_DEST)
    TKG_GOTO_DEST = \w[\w\d]* (IsPattern=Yes, Restricted=Yes)
    TKG_ARITH_BINARY_INT_DIVIDE = DIV:[\s(] (IsPattern=Yes)
    TKG_ARITH_BINARY_MODULO = MOD:[\s(] (IsPattern=Yes)
    TKG_FOR = FOR:\s (FileXLInvalid=Yes, IsPattern=Yes)
    TKG_ENDFOR = ENDFOR:[\s\n] (FileXLInvalid=Yes, IsPattern=Yes)
    TKG_FORTO = TO:\W (IsPattern=Yes)
    TKG_DO = repeat:[\s\n] (FileXLInvalid=Yes, IsPattern=Yes)
    TKG_ENDDO_UNTIL = until:[\s(] (FileXLInvalid=Yes, IsPattern=Yes)
    TKG_LOGICAL_UNARY_NOT = not:\W (IsPattern=Yes)
    TKG_SUPPRESS_SINGLE_STEP = NOHALT
    TKG_NC_BLOCK_PREFIX = N:[\s\d] (IsPattern=Yes)
    TKG_LOGICAL_HP_BINARY_AND = and:\W (IsPattern=Yes)
    TKG_LOGICAL_HP_BINARY_OR = or:\W (IsPattern=Yes)
    TKG_LOGICAL_HP_BINARY_XOR = xor:\W (IsPattern=Yes)
    TKG_BITWISE_BINARY_AND = b_and:\W (IsPattern=Yes)
    TKG_BITWISE_BINARY_OR = b_or:\W (IsPattern=Yes)
    TKG_BITWISE_BINARY_XOR = b_xor:\W (IsPattern=Yes)
    TKG_BITWISE_UNARY_COMPLEMENT = b_not:\W (IsPattern=Yes)
    TKG_IF = if:\W (FileXLInvalid=Yes, IsPattern=Yes)
    TKG_THEN = then:\W (FileXLInvalid=Yes, IsPattern=Yes)
    TKG_BLOCK_ELSE = else:\W (FileXLInvalid=Yes, IsPattern=Yes)
    TKG_BLOCK_ENDIF = endif:\W (FileXLInvalid=Yes, IsPattern=Yes)
    TKG_SWITCH = case:\W (FileXLInvalid=Yes, IsPattern=Yes)
    TKG_SWITCH_OF = of:\W (FileXLInvalid=Yes, IsPattern=Yes)
    TKG_SWITCH_DEFAULT = default:\W (FileXLInvalid=Yes, IsPattern=Yes)
    TKG_WHILE = while:\W (FileXLInvalid=Yes, IsPattern=Yes)
    TKG_ENDWHILE = endwhile (FileXLInvalid=Yes)
    TKG_FOREVER = loop:\W (FileXLInvalid=Yes, IsPattern=Yes)
    TKG_ENDFOREVER = endloop:\W (FileXLInvalid=Yes, IsPattern=Yes)
    TKG_LABEL_DEF = \w:\:|\w[\w\d]+:\: (IsPattern=Yes, FollowedBy=TKG_LABEL_SUFFIX)
    TKG_LABEL_SUFFIX = : (Restricted=Yes)
    TKG_MACRO_TEXT = . (Restricted=Yes, IsPattern=Yes)
    TKG_MACRO_NAME = [$\w][$\w\d(]+ (Restricted=Yes, IsPattern=Yes)
    TKG_PRIM_TYPE (IsPattern=Yes)
    TKG_OPEN_BRACKET = (
    TKG_CLOSE_BRACKET = )
    TKG_OPEN_INDEXBRACKET = [
    TKG_CLOSE_INDEXBRACKET = ]
    TKG_COMMA = ,
    TKG_DOT = \.:\w (IsPattern=Yes, FollowedBy=TKG_STRUCT_MEMBER_REF)
    TKG_STRUCT_MEMBER_REF = \w|\w[\w\d]+ (IsPattern=Yes, Restricted=Yes)
    TKG_PARAM_PREFIX = R:[\[\d]|$[RP]:[\[\d]|M[WLF]:[\[\d]|EX[WLBF]:[\[\d] (IsPattern=Yes)
    TKG_SUBRANGE = ..
    TKG_NUMBER = \d+\.\d+|\d+\.:[^\.] (IsPattern=Yes)
    TKG_INTEGER = \d+ (IsPattern=Yes)
    TKG_FRACTION = \.\d+ (IsPattern=Yes)
    TKG_NUMBER_EXP = EX:[\s\d\+\-\.] (IsPattern=Yes)
    TKG_STRING_CONCAT = <<
    TKG_COMP_BINARY_GREATER_THAN_OR_EQ = >=
    TKG_COMP_BINARY_LESS_THAN_OR_EQ = <=
    TKG_COMP_BINARY_EQUAL_TO = ==
    TKG_COMP_BINARY_NOT_EQUAL_TO = <>
    TKG_COMP_BINARY_GREATER_THAN = >
    TKG_COMP_BINARY_LESS_THAN = <
    TKG_ASSIGN_INCR = =ic:( (IsPattern=Yes)
    TKG_ASSIGN_EQ = =
    TKG_ARITH_BINARY_PLUS = +
    TKG_ARITH_BINARY_MINUS = -
    TKG_ARITH_BINARY_MULTIPLY = *
    TKG_ARITH_BINARY_DIVIDE = /
    TKG_SUBCALL_REPEAT_PREFIX = P:[\s\d] (IsPattern=Yes, FollowedBy=TKG_INTEGER)
    TKG_PV_DECL_REF = \w[\w\d\.\:\*]* (IsPattern=Yes, Restricted=Yes)
    TKG_G_CODE_PREFIX = G:[\s\d] (IsPattern=Yes)
    TKG_M_CODE_PREFIX = M:[\s\d(] (IsPattern=Yes)
    TKG_FUB_DECL = fub\s (IsPattern=Yes)
    TKG_FUB_ERR_LEV_1 = error_level_1:\s (IsPattern=Yes)
    TKG_FUB_ERR_LEV_2 = error_level_2:\s (IsPattern=Yes)
    TKG_FUB_ERR_LEV_3 = error_level_3:\s (IsPattern=Yes)
    TKG_FUB_ERR_LEV_4 = error_level_4:\s (IsPattern=Yes)
    TKG_FUB_BLOCKING = blocking:[\s\n] (IsPattern=Yes)
    TKG_FUB_NON_BLOCKING = non_blocking:\s (IsPattern=Yes)
    TKG_IEC_TYPED_VALUE = #[\w\d]+:[^\w\d\:] (IsPattern=Yes)
    TKG_REFERENCE = ref:[\s\n]|reference:[\s\n] (IsPattern=Yes, FollowedBy=TKG_IEC_TO)
    TKG_IEC_TO = to:[\s\n] (IsPattern=Yes, Restricted=Yes)
    TKG_ACCESS = ACCESS:[\s\n] (IsPattern=Yes)
    TKG_BINARY_LITERAL_START = 'B:[01_] (FollowedBy=TKG_BINARY_LITERAL_BODY, IsPattern=Yes)
    TKG_BINARY_LITERAL_BODY = [01_]+' (Restricted=Yes, IsPattern=Yes)
    TKG_HEX_LITERAL_START = 'H:[\dA-F_] (FollowedBy=TKG_HEX_LITERAL_BODY, IsPattern=Yes)
    TKG_HEX_LITERAL_BODY = [\dA-F_]+' (Restricted=Yes, IsPattern=Yes)
    TKG_WORD = \w|\w[\w\d\./]+|\./\w|\./\w[\w\d\./]+|[\^#][\w\d]+\:[\w\d\./]+ (IsPattern=Yes)
  StringChars (AsciiStringStart=", AsciiStringEnd=", UTF16StringStart=W", UTF16StringEnd=")
    EscapeSeq (Search=$N, ReplaceValue=10)
    EscapeSeq (Search=$L, ReplaceValue=10)
    EscapeSeq (Search=$P, ReplaceValue=12)
    EscapeSeq (Search=$R, ReplaceValue=13)
    EscapeSeq (Search=$T, ReplaceValue=9)
    EscapeSeq (Search=$Q, ReplaceStr=")
    EscapeSeq (Search=$', ReplaceStr=')
    EscapeSeq (Search=$", ReplaceStr=")
    EscapeSeq (Search=$[\dA-Fa-f]+, IsPattern=Yes, ReplaceEncodingBase=16)
    EscapeSeq (Search=$$, ReplaceStr=$)
    EscapeSeq (Search=$, ReplaceStr=)
```

### Data object Logical/GmcIpConfig/gmcipcsm (Cnc, version 3.14.3)

#### gmcipcsm.cnc
```
Root (LangModule=ailgcode, Version=1.0)
  Constants:
    NumAxes = 15 (Type=INT)
  Preprocess:
    PP_RULE_STOPRE (Search=STOPRE, Replace=G172)
    PP_RULE_CIP (Search=CIP:\W, Replace=G102, IsPattern=Yes)
  Types:
    RotationAngleSpecifier (type=ENUM, EnumType=REGEXP, Value6=H)
    RadiusSpecifier (type=ENUM, EnumType=REGEXP, Value1=R\s*=, Value2=CR\s*=)
    InterpolParam (type=ENUM, EnumType=REGEXP, Value0=I, Value1=J, Value2=K, Value100=G161\s*I, Value101=G161\s*J, Value102=G161\s*K, Value200=G162\s*I, Value201=G162\s*J, Value202=G162\s*K, Value0300=I\s*=\s*AC, Value0301=J\s*=\s*AC, Value0302=K\s*=\s*AC, Value0400=I\s*=\s*IC, Value0401=J\s*=\s*IC, Value0402=K\s*=\s*IC)
    CirclePointParam (type=ENUM, EnumType=REGEXP, Value0=I1\s*=, Value1=J1\s*=, Value2=K1\s*=, Value100=G161\s*I1\s*=, Value101=G161\s*J1\s*=, Value102=G161\s*K1\s*=, Value200=G162\s*I1\s*=, Value201=G162\s*J1\s*=, Value202=G162\s*K1\s*=, Value0300=I1\s*=\s*AC, Value0301=J1\s*=\s*AC, Value0302=K1\s*=\s*AC, Value0400=I1\s*=\s*IC, Value0401=J1\s*=\s*IC, Value0402=K1\s*=\s*IC)
    RPYAngleName (type=ENUM, EnumType=REGEXP, Value1=ROLL, Value0=PITCH, Value2=YAW)
    EulerAngleName (type=ENUM, EnumType=REGEXP, Value3=PHI, Value4=THETA, Value5=PSI)
    RotaryVectorName (type=ENUM, EnumType=REGEXP, Value0=P\s*=, Value1=Q\s*=, Value2=R\s*=)
    DwellTime (type=FLOAT)
    RParamIndex (type=INT, MinValue=0, MaxValue=999)
    EXParamIndex (type=INT, MinValue=0, MaxValue=99)
    MParamIndex (type=INT, MinValue=0, MaxValue=99)
    Byte (type=INT, MinValue=0, MaxValue=255)
    Word (type=INT, MinValue=-32768, MaxValue=32767)
    Long (type=INT)
  PVMacros:
    SAVE (ArrayDims=0, Group=500)
      CALL = Info(:id:52101, msg:"Save Modal GCode State NOT SUPPORTED YET":);
  SysVars
  Parameters:
    R (IndexType=RParamIndex, ValueType=FLOAT)
      ARG (ref=EXPR, DataType=RParamIndex)
    QUOTED (QuotedName=$R, Synchronous=Yes, IndexType=RParamIndex, ValueType=FLOAT)
      ARG (ref=EXPR, DataType=RParamIndex)
    QUOTED (QuotedName=$P, Synchronous=Yes, IndexType=RParamIndex, ValueType=FLOAT)
      ARG (ref=EXPR, DataType=RParamIndex)
    EXB (IndexType=EXParamIndex, ValueType=Byte)
      ARG (ref=EXPR, DataType=EXParamIndex)
    EXW (IndexType=EXParamIndex, ValueType=Word)
      ARG (ref=EXPR, DataType=EXParamIndex)
    EXL (IndexType=EXParamIndex, ValueType=Long)
      ARG (ref=EXPR, DataType=EXParamIndex)
    EXF (IndexType=EXFParamIndex, ValueType=FLOAT)
      ARG (ref=EXPR, DataType=EXFParamIndex)
    MW (Synchronous=Yes, IndexType=MParamIndex, ValueType=Word)
      ARG (ref=EXPR, DataType=MParamIndex)
    ML (Synchronous=Yes, IndexType=MParamIndex, ValueType=Long)
      ARG (ref=EXPR, DataType=MParamIndex)
    MF (Synchronous=Yes, IndexType=MParamIndex, ValueType=FLOAT)
      ARG (ref=EXPR, DataType=MParamIndex)
  MCodes:
    M17 = 17 (Group=41, Alias=RET:[^\d\w\(], Eval=Early, Inline=Yes, AliasIsPattern=Yes)
      ARG (ref=VALUE, DataType=FLOAT, RequireLiteral=Yes)
    M17_1 = 17.1 (Group=41, Alias=CONDRET, Eval=Early, Inline=Yes)
      ARG (ref=VALUE, DataType=FLOAT, RequireLiteral=Yes)
```

### Data object Logical/GmcIpConfig/gmcipcfg (Cnc)

#### gmcipcfg.cnc
```
CONFIG:
  LANG_INCLUDE gmcipmxd (LangName=IEC-ST, DataObject=Yes, IfNotExist=Error, Scope=NC_GLOBAL, RequireFnIgnore=MXConvertOrient)
  XML_INCLUDE gmcipvar (IfNotExist=Warn)
  XML_INCLUDE gmcipfun (IfNotExist=Warn)
  XML_INCLUDE gmcipfub (IfNotExist=Warn)
  MPQUEUE (NumPackets=200, LookaheadMinBlocks=5, LookaheadMaxBlocks=20, LookaheadMode=any, MaxPathJobs=256, CheckForNaNs=1)
  MONITOR (MaxPathStackEvents=1024)
  MPLOG (MaxBuffers=10, MinBuffers=4, EarlyCircleBufferLookahead=2, DefaultBufferSize=131072, TaskCycleDelay=1, FileDevice=mplog*, MaxLogFiles=20, MaxLogFileSize=1048576, CopyLineTextMaxChars=80)
  AXES (StandardCNCAxes=Yes)
  FUBOutputs:
    FUBOutput PLCOpen:
      ERROR (condition=$Error == 1)
      BUSY (condition=$Busy == 1)
    FUBOutput BuR:
      ERROR (condition=$status != 65535 && $status != 0)
      BUSY (condition=$status == 65535)
  FUNCTIONS:
    FUNC LEN (DeclareName=__LEN, AlwaysDeclare=Yes, RetType=INT)
      ARG IN (Type=STRING)
    FUNC LEFT (DeclareName=__LEFT, AlwaysDeclare=Yes, RetType=STRING, RetRef=Yes)
      ARG IN (Type=STRING)
      ARG L (Type=INT)
    FUNC RIGHT (DeclareName=__RIGHT, AlwaysDeclare=Yes, RetType=STRING, RetRef=Yes)
      ARG IN (Type=STRING)
      ARG L (Type=INT)
    FUNC MID (DeclareName=__MID, AlwaysDeclare=Yes, RetType=STRING, RetRef=Yes)
      ARG IN (Type=STRING)
      ARG L (Type=INT)
      ARG P (Type=INT)
    FUNC CONCAT (DeclareName=__CONCAT, AlwaysDeclare=Yes, RetType=STRING, RetRef=Yes)
      ARG IN1 (Type=STRING)
      ARG IN2 (Type=STRING)
    FUNC INSERT (DeclareName=__INSERT, AlwaysDeclare=Yes, RetType=STRING, RetRef=Yes)
      ARG IN1 (Type=STRING)
      ARG IN2 (Type=STRING)
      ARG P (Type=INT)
    FUNC DELETE (DeclareName=__DELETE, AlwaysDeclare=Yes, RetType=STRING, RetRef=Yes)
      ARG IN (Type=STRING)
      ARG L (Type=INT)
      ARG P (Type=INT)
    FUNC REPLACE (DeclareName=__REPLACE, AlwaysDeclare=Yes, RetType=STRING, RetRef=Yes)
      ARG IN1 (Type=STRING)
      ARG IN2 (Type=STRING)
      ARG L (Type=INT)
      ARG P (Type=INT)
    FUNC FIND (DeclareName=__FIND, AlwaysDeclare=Yes, RetType=INT)
      ARG IN1 (Type=STRING)
      ARG IN2 (Type=STRING)
  XML_INCLUDE gmcipuc (IfNotExist=Warn)
```

### Data object Logical/GmcIpConfig/gmcipiec (Cnc, version 3.14.3)

#### gmcipiec.cnc
```
Root (LangModule=ailgcode, Version=1.0)
  AxesSpec
  PrimTypes (PatternSuffix=:[^\d\w$#])
    BOOL (BRType=BOOL)
    STRING (BRType=STRING)
    WSTRING (BRType=WSTRING)
    TIME (BRType=TIME)
    SINT (BRType=SINT)
    INT (BRType=INT)
    DINT (BRType=DINT)
    USINT (BRType=USINT)
    UINT (BRType=UINT)
    UDINT (BRType=UDINT)
    REAL (BRType=REAL)
    LREAL (BRType=LREAL)
    DATE (BRType=DATE)
    DATE_AND_TIME (BRType=DATE_AND_TIME)
    DT (BRType=DT)
    TIME_OF_DAY (BRType=TIME_OF_DAY)
    TOD (BRType=TIME_OF_DAY)
    BYTE (BRType=BYTE)
    WORD (BRType=WORD)
    DWORD (BRType=DWORD)
  BuiltInProcs:
    SetCyclicId = #job->group_id = $[1]; (MinArgs=1, MaxArgs=1, Eval=Early)
    WaitForCyclic = if ( Defined(:$[1]:) ) 
        WaitForCyclicGroups(:${*}:);  
      else
        WaitForCyclicJob(:#last_job_id:);
      endif (MinArgs=0, MaxArgs=*)
    REPORT (MinArgs=2, MaxArgs=2)
      Arg (ref=id, DataType=INT)
      Arg (ref=msg, DataType=STRING)
    WARN (MinArgs=2, MaxArgs=2)
      Arg (ref=id, DataType=INT)
      Arg (ref=msg, DataType=STRING)
    HALT (MinArgs=2, MaxArgs=2)
      Arg (ref=id, DataType=INT)
      Arg (ref=msg, DataType=STRING)
    ERROR (MinArgs=2, MaxArgs=2)
      Arg (ref=id, DataType=INT)
      Arg (ref=msg, DataType=STRING)
    LOADBG (MinArgs=1, MaxArgs=1)
      Arg (ref=filename, DataType=STRING)
    LOAD (MinArgs=1, MaxArgs=1)
      Arg (ref=filename, DataType=STRING)
    UNLOAD (MinArgs=1, MaxArgs=1)
      Arg (ref=filename, DataType=STRING)
    EXEC (MinArgs=1, MaxArgs=5)
      Arg (ref=filename, DataType=STRING)
      Arg (ref=arguments, DataType=ANY_DATA)
      Arg (ref=langId, DataType=INT)
      Arg (ref=block, DataType=INT, MinCount=0, MaxCount=1, DenyArgs=5, WriteOpts=:)
      Arg (ref=line, DataType=INT, MinCount=0, MaxCount=1, DenyArgs=4, WriteOpts=:)
    EXEC_RPC (MinArgs=2, MaxArgs=4)
      Arg (ref=filename, DataType=STRING)
      Arg (ref=arguments, DataType=ANY_DATA)
      Arg (ref=langId, DataType=INT)
      Arg (ref=rpc, DataType=ANY_DATA, MinCount=1, MaxCount=1)
    EVAL (MinArgs=1, MaxArgs=2)
      Arg (ref=expression, DataType=STRING)
      Arg (ref=langId, DataType=INT)
    PUSH_PACKET = PushPacket(::);
    PUSH_PACKET_CMD (MinArgs=1, MaxArgs=2)
      Arg (ref=cmd, DataType=INT)
      Arg (ref=data, DataType=ANY_DATA)
    DISPATCH_AND_WAIT (MinArgs=1, MaxArgs=1)
      Arg (ref=cmd, DataType=INT)
    START_PACKET_LIST = #inhibit_mp_list_dispatch = 1;
    END_PACKET_LIST = #inhibit_mp_list_dispatch = 0;
    LOG_INFO (MinArgs=1, MaxArgs=1)
      Arg (ref=msg, DataType=STRING)
    SET_BLOCK_NUMBER = SetCurBlockNr(:$[1]:); (MinArgs=1, MaxArgs=1)
    SBLOF_PATH = #next_motion.Command = MPCMD_SBL_PATH_INHIBIT;
      PushPacket(::);
    SBLON_PATH = #next_motion.Command = MPCMD_SBL_PATH_RELEASE;
      PushPacket(::);
  BuiltInFns:
    ABS = Abs(:$[1]:) (ReturnType=ANY_NUM, ArgType1=ANY_NUM, Inline=Yes)
    SIN = RSin(:$[1]:) (ReturnType=ANY_REAL, ArgType1=ANY_REAL, Inline=Yes)
    COS = RCos(:$[1]:) (ReturnType=ANY_REAL, ArgType1=ANY_REAL, Inline=Yes)
    TAN = RTan(:$[1]:) (ReturnType=ANY_REAL, ArgType1=ANY_REAL, Inline=Yes)
    ASIN = RASin(:$[1]:) (ReturnType=ANY_REAL, ArgType1=ANY_REAL, Inline=Yes)
    ACOS = RACos(:$[1]:) (ReturnType=ANY_REAL, ArgType1=ANY_REAL, Inline=Yes)
    ATAN = RATan(:$[1]:) (ReturnType=ANY_REAL, ArgType1=ANY_REAL, Inline=Yes)
    SQRT = Sqrt(:$[1]:) (ReturnType=ANY_REAL, ArgType1=ANY_REAL, Inline=Yes)
    LN = Ln(:$[1]:) (ReturnType=ANY_REAL, ArgType1=ANY_REAL, Inline=Yes)
    EXP = Exp(:$[1]:) (ReturnType=ANY_REAL, ArgType1=ANY_REAL, Inline=Yes)
    LOG = Log(:$[1]:) (ReturnType=ANY_REAL, ArgType1=ANY_REAL, Inline=Yes)
    EXPT = Pow(:$[1],$[2]:) (ReturnType=ANY_REAL, ArgType1=ANY_REAL, ArgType2=ANY_NUM, Inline=Yes)
    TRUNC = ToInt(:Fix(:$[1]:):) (ReturnType=IEC_INT, ArgType1=FLOAT, Inline=Yes)
    ADR = Adr(:\$[1]:) (ReturnType=IEC_UDINT, ArgType1=ANY_DATA, Inline=Yes)
    REF = \$[1] (ReturnType=ANY_DATA, ArgType1=ANY_DATA, Inline=Yes)
    SIZEOF = Sizeof(:\$[1]:) (ReturnType=IEC_UINT, NumArgs=1, Inline=Yes)
    LIMIT (ReturnType=ANY_NUM, Inline=No)
      Arg (ref=MIN, DataType=ANY_NUM)
      Arg (ref=IN, DataType=ANY_NUM)
      Arg (ref=MAX, DataType=ANY_NUM)
    MIN (ReturnType=ANY_NUM, Inline=No)
      Arg (ref=IN1, DataType=ANY_NUM)
      Arg (ref=IN2, DataType=ANY_NUM)
    MAX (ReturnType=ANY_NUM, Inline=No)
      Arg (ref=IN1, DataType=ANY_NUM)
      Arg (ref=IN2, DataType=ANY_NUM)
    ROL = BitRotL(:$[1],$[2]:) (ReturnType=ANY_NUM, ArgType1=ANY_NUM, ArgType2=IEC_SINT)
    ROR = BitRotR(:$[1],$[2]:) (ReturnType=ANY_NUM, ArgType1=ANY_NUM, ArgType2=IEC_SINT)
    SHR = BitShR(:$[1],$[2]:) (ReturnType=ANY_NUM, ArgType1=ANY_NUM, ArgType2=IEC_SINT)
    SHL = BitShL(:$[1],$[2]:) (ReturnType=ANY_NUM, ArgType1=ANY_NUM, ArgType2=IEC_SINT)
    BIT_TST = AsBitTst(:$[1],$[2]:) (ReturnType=ANY_NUM, ArgType1=ANY_NUM, ArgType2=IEC_SINT)
    BIT_SET = AsBitSet(:$[1],$[2]:) (ReturnType=ANY_NUM, ArgType1=ANY_NUM, ArgType2=IEC_SINT)
    BIT_CLR = AsBitClr(:$[1],$[2]:) (ReturnType=ANY_NUM, ArgType1=ANY_NUM, ArgType2=IEC_SINT)
    TO_BOOL = ToBool(:$[1]:) (ReturnType=IEC_BOOL, ArgType1=ANY_DATA, Inline=Yes)
    TO_USINT = ToUInt(:$[1],1:) (ReturnType=IEC_USINT, ArgType1=ANY_DATA, Inline=Yes)
    TO_BYTE = ToUInt(:$[1],1:) (ReturnType=IEC_BYTE, ArgType1=ANY_DATA, Inline=Yes)
    TO_SINT = ToInt(:$[1],1:) (ReturnType=IEC_SINT, ArgType1=ANY_DATA, Inline=Yes)
    TO_UINT = ToUInt(:$[1],2:) (ReturnType=IEC_UINT, ArgType1=ANY_DATA, Inline=Yes)
    TO_WORD = ToUInt(:$[1],2:) (ReturnType=IEC_WORD, ArgType1=ANY_DATA, Inline=Yes)
    TO_INT = ToInt(:$[1],2:) (ReturnType=IEC_INT, ArgType1=ANY_DATA, Inline=Yes)
    TO_UDINT = ToUInt(:$[1]:) (ReturnType=IEC_UDINT, ArgType1=ANY_DATA, Inline=Yes)
    TO_DWORD = ToUInt(:$[1]:) (ReturnType=IEC_DWORD, ArgType1=ANY_DATA, Inline=Yes)
    TO_DINT = ToInt(:$[1]:) (ReturnType=IEC_DINT, ArgType1=ANY_DATA, Inline=Yes)
    TO_TIME = ToTime(:$[1]:) (ReturnType=IEC_TIME, ArgType1=ANY_DATA, Inline=Yes)
    TO_DT = ToDT(:$[1]:) (ReturnType=IEC_DT, ArgType1=ANY_DATA, Inline=Yes)
    TO_DATE_AND_TIME = ToDT(:$[1]:) (ReturnType=IEC_DT, ArgType1=ANY_DATA, Inline=Yes)
    TO_TOD = ToTOD(:$[1]:) (ReturnType=IEC_TOD, ArgType1=ANY_DATA, Inline=Yes)
    TO_TIME_OF_DAY = ToTOD(:$[1]:) (ReturnType=IEC_TOD, ArgType1=ANY_DATA, Inline=Yes)
    TO_DATE = ToDate(:$[1]:) (ReturnType=IEC_DATE, ArgType1=ANY_DATA, Inline=Yes)
    TO_REAL = ToFloat(:$[1]:) (ReturnType=IEC_REAL, ArgType1=ANY_DATA, Inline=Yes)
    TO_LREAL = ToLReal(:$[1]:) (ReturnType=IEC_LREAL, ArgType1=ANY_DATA, Inline=Yes)
    TO_STRING = ToString(:$[1]:) (ReturnType=IEC_STRING, ArgType1=ANY_DATA, Inline=Yes)
    TO_WSTRING = ToWString(:$[1]:) (ReturnType=IEC_WSTRING, ArgType1=ANY_DATA, Inline=Yes)
    USINT_TO_BOOL = ToBool(:$[1]:) (ReturnType=IEC_BOOL, ArgType1=IEC_USINT, Inline=Yes)
    SINT_TO_BOOL = ToBool(:$[1]:) (ReturnType=IEC_BOOL, ArgType1=IEC_SINT, Inline=Yes)
    UINT_TO_BOOL = ToBool(:$[1]:) (ReturnType=IEC_BOOL, ArgType1=IEC_UINT, Inline=Yes)
    INT_TO_BOOL = ToBool(:$[1]:) (ReturnType=IEC_BOOL, ArgType1=IEC_INT, Inline=Yes)
    UDINT_TO_BOOL = ToBool(:$[1]:) (ReturnType=IEC_BOOL, ArgType1=IEC_UDINT, Inline=Yes)
    DINT_TO_BOOL = ToBool(:$[1]:) (ReturnType=IEC_BOOL, ArgType1=IEC_DINT, Inline=Yes)
    REAL_TO_BOOL = ToBool(:$[1]:) (ReturnType=IEC_BOOL, ArgType1=IEC_REAL, Inline=Yes)
    LREAL_TO_BOOL = ToBool(:$[1]:) (ReturnType=IEC_BOOL, ArgType1=IEC_LREAL, Inline=Yes)
    TIME_TO_BOOL = ToBool(:$[1]:) (ReturnType=IEC_BOOL, ArgType1=IEC_TIME, Inline=Yes)
    DT_TO_BOOL = ToBool(:$[1]:) (ReturnType=IEC_BOOL, ArgType1=IEC_DT, Inline=Yes)
    TOD_TO_BOOL = ToBool(:$[1]:) (ReturnType=IEC_BOOL, ArgType1=IEC_TOD, Inline=Yes)
    BYTE_TO_BOOL = ToBool(:$[1]:) (ReturnType=IEC_BOOL, ArgType1=IEC_BYTE, Inline=Yes)
    WORD_TO_BOOL = ToBool(:$[1]:) (ReturnType=IEC_BOOL, ArgType1=IEC_WORD, Inline=Yes)
    DWORD_TO_BOOL = ToBool(:$[1]:) (ReturnType=IEC_BOOL, ArgType1=IEC_DWORD, Inline=Yes)
    BOOL_TO_USINT = ToUInt(:$[1],1:) (ReturnType=IEC_USINT, ArgType1=IEC_BOOL, Inline=Yes)
    SINT_TO_USINT = ToUInt(:$[1],1:) (ReturnType=IEC_USINT, ArgType1=IEC_SINT, Inline=Yes)
    UINT_TO_USINT = ToUInt(:$[1],1:) (ReturnType=IEC_USINT, ArgType1=IEC_UINT, Inline=Yes)
    INT_TO_USINT = ToUInt(:$[1],1:) (ReturnType=IEC_USINT, ArgType1=IEC_INT, Inline=Yes)
    UDINT_TO_USINT = ToUInt(:$[1],1:) (ReturnType=IEC_USINT, ArgType1=IEC_UDINT, Inline=Yes)
    DINT_TO_USINT = ToUInt(:$[1],1:) (ReturnType=IEC_USINT, ArgType1=IEC_DINT, Inline=Yes)
    REAL_TO_USINT = ToUInt(:$[1],1:) (ReturnType=IEC_USINT, ArgType1=IEC_REAL, Inline=Yes)
    LREAL_TO_USINT = ToUInt(:$[1],1:) (ReturnType=IEC_USINT, ArgType1=IEC_LREAL, Inline=Yes)
    BOOL_TO_SINT = ToInt(:$[1],1:) (ReturnType=IEC_SINT, ArgType1=IEC_BOOL, Inline=Yes)
    USINT_TO_SINT = ToInt(:$[1],1:) (ReturnType=IEC_SINT, ArgType1=IEC_USINT, Inline=Yes)
    UINT_TO_SINT = ToInt(:$[1],1:) (ReturnType=IEC_SINT, ArgType1=IEC_UINT, Inline=Yes)
    INT_TO_SINT = ToInt(:$[1],1:) (ReturnType=IEC_SINT, ArgType1=IEC_INT, Inline=Yes)
    UDINT_TO_SINT = ToInt(:$[1],1:) (ReturnType=IEC_SINT, ArgType1=IEC_UDINT, Inline=Yes)
    DINT_TO_SINT = ToInt(:$[1],1:) (ReturnType=IEC_SINT, ArgType1=IEC_DINT, Inline=Yes)
    REAL_TO_SINT = ToInt(:$[1],1:) (ReturnType=IEC_SINT, ArgType1=IEC_REAL, Inline=Yes)
    LREAL_TO_SINT = ToInt(:$[1],1:) (ReturnType=IEC_SINT, ArgType1=IEC_LREAL, Inline=Yes)
    BOOL_TO_UINT = ToUInt(:$[1],2:) (ReturnType=IEC_UINT, ArgType1=IEC_BOOL, Inline=Yes)
    SINT_TO_UINT = ToUInt(:$[1],2:) (ReturnType=IEC_UINT, ArgType1=IEC_SINT, Inline=Yes)
    USINT_TO_UINT = ToUInt(:$[1],2:) (ReturnType=IEC_UINT, ArgType1=IEC_USINT, Inline=Yes)
    INT_TO_UINT = ToUInt(:$[1],2:) (ReturnType=IEC_UINT, ArgType1=IEC_INT, Inline=Yes)
    UDINT_TO_UINT = ToUInt(:$[1],2:) (ReturnType=IEC_UINT, ArgType1=IEC_UDINT, Inline=Yes)
    DINT_TO_UINT = ToUInt(:$[1],2:) (ReturnType=IEC_UINT, ArgType1=IEC_DINT, Inline=Yes)
    REAL_TO_UINT = ToUInt(:$[1],2:) (ReturnType=IEC_UINT, ArgType1=IEC_REAL, Inline=Yes)
    LREAL_TO_UINT = ToUInt(:$[1],2:) (ReturnType=IEC_UINT, ArgType1=IEC_LREAL, Inline=Yes)
    BOOL_TO_INT = ToInt(:$[1],2:) (ReturnType=IEC_INT, ArgType1=IEC_BOOL, Inline=Yes)
    SINT_TO_INT = ToInt(:$[1],2:) (ReturnType=IEC_INT, ArgType1=IEC_SINT, Inline=Yes)
    USINT_TO_INT = ToInt(:$[1],2:) (ReturnType=IEC_INT, ArgType1=IEC_USINT, Inline=Yes)
    UINT_TO_INT = ToInt(:$[1],2:) (ReturnType=IEC_INT, ArgType1=IEC_UINT, Inline=Yes)
    UDINT_TO_INT = ToInt(:$[1],2:) (ReturnType=IEC_INT, ArgType1=IEC_UDINT, Inline=Yes)
    DINT_TO_INT = ToInt(:$[1],2:) (ReturnType=IEC_INT, ArgType1=IEC_DINT, Inline=Yes)
    REAL_TO_INT = ToInt(:$[1],2:) (ReturnType=IEC_INT, ArgType1=IEC_REAL, Inline=Yes)
    LREAL_TO_INT = ToInt(:$[1],2:) (ReturnType=IEC_INT, ArgType1=IEC_LREAL, Inline=Yes)
    BOOL_TO_UDINT = ToUInt(:$[1]:) (ReturnType=IEC_UDINT, ArgType1=IEC_BOOL, Inline=Yes)
    USINT_TO_UDINT = ToUInt(:$[1]:) (ReturnType=IEC_UDINT, ArgType1=IEC_USINT, Inline=Yes)
    SINT_TO_UDINT = ToUInt(:$[1]:) (ReturnType=IEC_UDINT, ArgType1=IEC_SINT, Inline=Yes)
    UINT_TO_UDINT = ToUInt(:$[1]:) (ReturnType=IEC_UDINT, ArgType1=IEC_UINT, Inline=Yes)
    INT_TO_UDINT = ToUInt(:$[1]:) (ReturnType=IEC_UDINT, ArgType1=IEC_INT, Inline=Yes)
    DINT_TO_UDINT = ToUInt(:$[1]:) (ReturnType=IEC_UDINT, ArgType1=IEC_DINT, Inline=Yes)
    REAL_TO_UDINT = ToUInt(:$[1]:) (ReturnType=IEC_UDINT, ArgType1=IEC_REAL, Inline=Yes)
    LREAL_TO_UDINT = ToUInt(:$[1]:) (ReturnType=IEC_UDINT, ArgType1=IEC_LREAL, Inline=Yes)
    TIME_TO_UDINT = ToUInt(:$[1]:) (ReturnType=IEC_UDINT, ArgType1=IEC_TIME, Inline=Yes)
    DT_TO_UDINT = ToUInt(:$[1]:) (ReturnType=IEC_UDINT, ArgType1=IEC_DT, Inline=Yes)
    BOOL_TO_DINT = ToInt(:$[1]:) (ReturnType=IEC_DINT, ArgType1=IEC_BOOL, Inline=Yes)
    USINT_TO_DINT = ToInt(:$[1]:) (ReturnType=IEC_DINT, ArgType1=IEC_USINT, Inline=Yes)
    SINT_TO_DINT = ToInt(:$[1]:) (ReturnType=IEC_DINT, ArgType1=IEC_SINT, Inline=Yes)
    UINT_TO_DINT = ToInt(:$[1]:) (ReturnType=IEC_DINT, ArgType1=IEC_UINT, Inline=Yes)
    INT_TO_DINT = ToInt(:$[1]:) (ReturnType=IEC_DINT, ArgType1=IEC_INT, Inline=Yes)
    UDINT_TO_DINT = ToInt(:$[1]:) (ReturnType=IEC_DINT, ArgType1=IEC_UDINT, Inline=Yes)
    REAL_TO_DINT = ToInt(:$[1]:) (ReturnType=IEC_DINT, ArgType1=IEC_REAL, Inline=Yes)
    LREAL_TO_DINT = ToInt(:$[1]:) (ReturnType=IEC_DINT, ArgType1=IEC_LREAL, Inline=Yes)
    TIME_TO_DINT = ToInt(:$[1]:) (ReturnType=IEC_DINT, ArgType1=IEC_TIME, Inline=Yes)
    DT_TO_DINT = ToInt(:$[1]:) (ReturnType=IEC_DINT, ArgType1=IEC_DT, Inline=Yes)
    BOOL_TO_TIME = ToTime(:$[1]:) (ReturnType=IEC_TIME, ArgType1=IEC_BOOL, Inline=Yes)
    DINT_TO_TIME = ToTime(:$[1]:) (ReturnType=IEC_TIME, ArgType1=IEC_DINT, Inline=Yes)
    UDINT_TO_TIME = ToTime(:$[1]:) (ReturnType=IEC_TIME, ArgType1=IEC_UDINT, Inline=Yes)
    BOOL_TO_DT = ToDT(:$[1]:) (ReturnType=IEC_DT, ArgType1=IEC_BOOL, Inline=Yes)
    DINT_TO_DT = ToDT(:$[1]:) (ReturnType=IEC_DT, ArgType1=IEC_DINT, Inline=Yes)
    UDINT_TO_DT = ToDT(:$[1]:) (ReturnType=IEC_DT, ArgType1=IEC_UDINT, Inline=Yes)
    BOOL_TO_REAL = ToFloat(:$[1]:) (ReturnType=IEC_REAL, ArgType1=IEC_BOOL, Inline=Yes)
    USINT_TO_REAL = ToFloat(:$[1]:) (ReturnType=IEC_REAL, ArgType1=IEC_USINT, Inline=Yes)
    SINT_TO_REAL = ToFloat(:$[1]:) (ReturnType=IEC_REAL, ArgType1=IEC_SINT, Inline=Yes)
    UINT_TO_REAL = ToFloat(:$[1]:) (ReturnType=IEC_REAL, ArgType1=IEC_UINT, Inline=Yes)
    INT_TO_REAL = ToFloat(:$[1]:) (ReturnType=IEC_REAL, ArgType1=IEC_INT, Inline=Yes)
    UDINT_TO_REAL = ToFloat(:$[1]:) (ReturnType=IEC_REAL, ArgType1=IEC_UDINT, Inline=Yes)
    DINT_TO_REAL = ToFloat(:$[1]:) (ReturnType=IEC_REAL, ArgType1=IEC_DINT, Inline=Yes)
    LREAL_TO_REAL = ToFloat(:$[1]:) (ReturnType=IEC_REAL, ArgType1=IEC_LREAL, Inline=Yes)
    TIME_TO_REAL = ToFloat(:$[1]:) (ReturnType=IEC_REAL, ArgType1=IEC_TIME, Inline=Yes)
    BOOL_TO_LREAL = ToLReal(:$[1]:) (ReturnType=IEC_LREAL, ArgType1=IEC_BOOL, Inline=Yes)
    USINT_TO_LREAL = ToLReal(:$[1]:) (ReturnType=IEC_LREAL, ArgType1=IEC_USINT, Inline=Yes)
    SINT_TO_LREAL = ToLReal(:$[1]:) (ReturnType=IEC_LREAL, ArgType1=IEC_SINT, Inline=Yes)
    UINT_TO_LREAL = ToLReal(:$[1]:) (ReturnType=IEC_LREAL, ArgType1=IEC_UINT, Inline=Yes)
    INT_TO_LREAL = ToLReal(:$[1]:) (ReturnType=IEC_LREAL, ArgType1=IEC_INT, Inline=Yes)
    UDINT_TO_LREAL = ToLReal(:$[1]:) (ReturnType=IEC_LREAL, ArgType1=IEC_UDINT, Inline=Yes)
    DINT_TO_LREAL = ToLReal(:$[1]:) (ReturnType=IEC_LREAL, ArgType1=IEC_DINT, Inline=Yes)
    REAL_TO_LREAL = ToLReal(:$[1]:) (ReturnType=IEC_LREAL, ArgType1=IEC_REAL, Inline=Yes)
    TIME_TO_LREAL = ToLReal(:$[1]:) (ReturnType=IEC_LREAL, ArgType1=IEC_TIME, Inline=Yes)
    BOOL_TO_STRING = ToString(:ToBool(:$[1]:):) (ReturnType=IEC_STRING, ArgType1=IEC_BOOL, Inline=Yes)
    USINT_TO_STRING = ToString(:ToUInt(:$[1],1:):) (ReturnType=IEC_STRING, ArgType1=IEC_USINT, Inline=Yes)
    SINT_TO_STRING = ToString(:ToInt(:$[1],1:):) (ReturnType=IEC_STRING, ArgType1=IEC_SINT, Inline=Yes)
    UINT_TO_STRING = ToString(:ToUInt(:$[1],2:):) (ReturnType=IEC_STRING, ArgType1=IEC_UINT, Inline=Yes)
    INT_TO_STRING = ToString(:ToInt(:$[1],2:):) (ReturnType=IEC_STRING, ArgType1=IEC_INT, Inline=Yes)
    UDINT_TO_STRING = ToString(:ToUInt(:$[1]:):) (ReturnType=IEC_STRING, ArgType1=IEC_UDINT, Inline=Yes)
    DINT_TO_STRING = ToString(:ToInt(:$[1]:):) (ReturnType=IEC_STRING, ArgType1=IEC_DINT, Inline=Yes)
    REAL_TO_STRING = ToString(:ToFloat(:$[1]:):) (ReturnType=IEC_STRING, ArgType1=IEC_REAL, Inline=Yes)
    LREAL_TO_STRING = ToString(:ToLReal(:$[1]:):) (ReturnType=IEC_STRING, ArgType1=IEC_LREAL, Inline=Yes)
    STRING_TO_BOOL = ToBool(:StrToInt(:$[1]:):) (ReturnType=IEC_BOOL, ArgType1=IEC_STRING, Inline=Yes)
    STRING_TO_USINT = ToUInt(:StrToInt(:$[1]:),1:) (ReturnType=IEC_USINT, ArgType1=IEC_STRING, Inline=Yes)
    STRING_TO_SINT = ToInt(:StrToInt(:$[1]:),1:) (ReturnType=IEC_SINT, ArgType1=IEC_STRING, Inline=Yes)
    STRING_TO_UINT = ToUInt(:StrToInt(:$[1]:),2:) (ReturnType=IEC_UINT, ArgType1=IEC_STRING, Inline=Yes)
    STRING_TO_INT = ToInt(:StrToInt(:$[1]:),2:) (ReturnType=IEC_INT, ArgType1=IEC_STRING, Inline=Yes)
    STRING_TO_UDINT = ToUInt(:StrToInt(:$[1]:):) (ReturnType=IEC_UDINT, ArgType1=IEC_STRING, Inline=Yes)
    STRING_TO_DINT = ToInt(:StrToInt(:$[1]:):) (ReturnType=IEC_DINT, ArgType1=IEC_STRING, Inline=Yes)
    STRING_TO_REAL = ToFloat(:ToLReal(:$[1]:):) (ReturnType=IEC_REAL, ArgType1=IEC_STRING, Inline=Yes)
    STRING_TO_LREAL = ToLReal(:$[1]:) (ReturnType=IEC_LREAL, ArgType1=IEC_STRING, Inline=Yes)
    LEN = __LEN(:$[1]:) (ReturnType=IEC_INT, ArgType1=IEC_STRING, Inline=Yes)
    LEFT = __LEFT(:$[1], $[2]:) (ReturnType=IEC_STRING, ArgType1=IEC_STRING, ArgType2=IEC_INT, Inline=Yes)
    RIGHT = __RIGHT(:$[1], $[2]:) (ReturnType=IEC_STRING, ArgType1=IEC_STRING, ArgType2=IEC_INT, Inline=Yes)
    MID = __MID(:$[1], $[2], $[3]:) (ReturnType=IEC_STRING, ArgType1=IEC_STRING, ArgType2=IEC_INT, ArgType3=IEC_INT, Inline=Yes)
    CONCAT = __CONCAT(:$[1], $[2]:) (ReturnType=IEC_STRING, ArgType1=IEC_STRING, ArgType2=IEC_STRING, Inline=Yes)
    INSERT = __INSERT(:$[1], $[2], $[3]:) (ReturnType=IEC_STRING, ArgType1=IEC_STRING, ArgType2=IEC_STRING, ArgType3=IEC_INT, Inline=Yes)
    DELETE = __DELETE(:$[1], $[2], $[3]:) (ReturnType=IEC_STRING, ArgType1=IEC_STRING, ArgType2=IEC_INT, ArgType3=IEC_INT, Inline=Yes)
    REPLACE = __REPLACE(:$[1], $[2], $[3], $[4]:) (ReturnType=IEC_STRING, ArgType1=IEC_STRING, ArgType2=IEC_STRING, ArgType3=IEC_INT, ArgType4=IEC_INT, Inline=Yes)
    FIND = __FIND(:$[1], $[2]:) (ReturnType=IEC_INT, ArgType1=IEC_STRING, ArgType2=IEC_STRING, Inline=Yes)
    IP_INST_NUM = IpInstNum(::) (ReturnType=IEC_INT, NumArgs=0)
    IP_OWNER_ID = IpOwnerId(::) (ReturnType=IEC_INT, NumArgs=0)
    PACKET_DATA_ADR = GetIpInt(:6:) (ReturnType=IEC_UDINT, NumArgs=0, Inline=Yes)
    PACKET_COMMAND_ADR = GetIpInt(:7:) (ReturnType=IEC_UDINT, NumArgs=0, Inline=Yes)
  Parameters:
    QUOTED (QuotedName=$R, ValueType=FLOAT, ReturnType=IEC_LREAL)
      ARG (ref=EXPR, DataType=INT, MinValue=0, MaxValue=999)
    QUOTED (QuotedName=$P, ValueType=FLOAT, ReturnType=IEC_LREAL)
      ARG (ref=EXPR, DataType=INT, MinValue=0, MaxValue=999)
    QUOTED (QuotedName=$EXB, ValueType=INT, ReturnType=IEC_SINT)
      ARG (ref=EXPR, DataType=INT, MinValue=0, MaxValue=99)
    QUOTED (QuotedName=$EXW, ValueType=INT, ReturnType=IEC_INT)
      ARG (ref=EXPR, DataType=INT, MinValue=0, MaxValue=99)
    QUOTED (QuotedName=$EXL, ValueType=INT, ReturnType=IEC_DINT)
      ARG (ref=EXPR, DataType=INT, MinValue=0, MaxValue=99)
    QUOTED (QuotedName=$EXF, ValueType=FLOAT, ReturnType=IEC_REAL)
      ARG (ref=EXPR, DataType=INT, MinValue=0, MaxValue=3999)
    QUOTED (QuotedName=$MW, Synchronous=Yes, ValueType=INT, ReturnType=IEC_INT)
      ARG (ref=EXPR, DataType=INT, MinValue=0, MaxValue=99)
    QUOTED (QuotedName=$ML, Synchronous=Yes, ValueType=INT, ReturnType=IEC_DINT)
      ARG (ref=EXPR, DataType=INT, MinValue=0, MaxValue=99)
    QUOTED (QuotedName=$MF, Synchronous=Yes, ValueType=FLOAT, ReturnType=IEC_REAL)
      ARG (ref=EXPR, DataType=INT, MinValue=0, MaxValue=99)
  ParserData (NestedComments=No, DefaultCaseSensitive=Yes, CommentsSpanLines=Yes, ReadWholeFileBeforeParsing=Yes, ExpectMainProgStmts=No, UseFubTemplates=No, LexerType=IEC, RuntimePreventOverflow=No, RoundRealToInt=No, AllowArrayRefWithoutIndex=Yes, DeclareEnumLiteralsAsConstants=No, AllowVariableAutoDereference=Yes, AllowStructMemberAutoDereference=No, AllowPassByRefFnArgAutoReference=No, AllowNamedFnArgs=Yes, AllowUnnamedFnArgs=Yes, AllowFnArgMixedNaming=Yes, AllowFnArgsOutOfSequence=No, AllowBuiltinFnArgsOutOfSequence=Yes, AllowFnArgsOmmitted=Yes, AllowIgnoredFnReturn=Yes, AllowIgnoredExtraSubArgs=No, AllowFnStringInputArgsShort=No, RefuseBuiltinFnUnknownArgName=Yes, AllowBuiltinFnArgCaseSensitive=Yes)
    TKG_OPEN_COMMENT = (*
    TKG_CLOSE_COMMENT = *)
    TKG_IEC_LINE_COMMENT = //
    TKG_TRUE = TRUE:[^\w\d] (IsPattern=Yes)
    TKG_FALSE = FALSE:[^\w\d] (IsPattern=Yes)
    TKG_PRIM_TYPE (IsPattern=Yes)
    TKG_OPEN_BRACKET = (
    TKG_CLOSE_BRACKET = )
    TKG_OPEN_INDEXBRACKET = [
    TKG_CLOSE_INDEXBRACKET = ]
    TKG_COMMA = ,
    TKG_SUBRANGE = ..
    TKG_IEC_BINARY_INTEGER = 2#_[01][01_]+|2#[01][01_]+|2#_[01]|2#[01] (IsPattern=Yes)
    TKG_IEC_OCTAL_INTEGER = 8#_[0-7][0-7_]+|8#[0-7][0-7_]+|8#_[0-7]|8#[0-7] (IsPattern=Yes)
    TKG_IEC_HEX_INTEGER = 16#_[\da-fA-F][\da-fA-F]+|16#[\da-fA-F][\da-fA-F_]+|16#_[\da-fA-F]|16#[\da-fA-F] (IsPattern=Yes)
    TKG_REAL = \d[\d_]*\.[\d_]+[Ee][\+\-]\d[\d_]*|\d[\d_]*\.[\d_]+[Ee]\d[\d_]*|\d[\d_]*\.[\d_]+ (IsPattern=Yes)
    TKG_REAL_EXP = \d[\d_]*[Ee]\d[\d_]*|\d[\d_]*[Ee][\+\-]\d[\d_]* (IsPattern=Yes)
    TKG_INTEGER = \d|\d[\d_]+ (IsPattern=Yes)
    TKG_DOT = .
    TKG_PATHSYNCH_REC_IEC = DO_PATH_SYNCH:[^\w\d] (IsPattern=Yes, EndRuleToken=Yes)
    TKG_PATHSYNCH_END = END_PATH_SYNCH:[^\w\d] (IsPattern=Yes, EndRuleToken=Yes)
    TKG_PATHSYNCH_IPEVAL = IP_EVAL:[^\w\d] (IsPattern=Yes)
    TKG_CYCLIC_PATHSYNCH_BLOCKING_IEC = CYCLIC_PS_BL:[^\w\d] (IsPattern=Yes, EndRuleToken=Yes)
    TKG_CYCLIC_PATHSYNCH_IEC = CYCLIC_PS:[^\w\d] (IsPattern=Yes, EndRuleToken=Yes)
    TKG_CYCLIC_BLOCKING_IEC = CYCLIC_BL:[^\w\d] (IsPattern=Yes, EndRuleToken=Yes)
    TKG_CYCLIC_IEC = CYCLIC:[^\w\d] (IsPattern=Yes, EndRuleToken=Yes)
    TKG_CYCLIC_END_IEC = END_CYCLIC:[^\w\d] (IsPattern=Yes, EndRuleToken=Yes)
    TKG_REFERENCE = REFERENCE:[^\w\d] (FollowedBy=TKG_IEC_TO, IsPattern=Yes)
    TKG_IEC_TO = TO:[^\w\d] (IsPattern=Yes)
    TKG_IEC_DO = DO:[^\w\d] (IsPattern=Yes, EndRuleToken=Yes)
    TKG_FOR_NOFINALDEC = FOR:[^\w\d] (FileXLInvalid=Yes, IsPattern=Yes)
    TKG_FORSTEP = BY:[^\w\d] (FileXLInvalid=Yes, IsPattern=Yes)
    TKG_ENDFOR = END_FOR:[^\w\d] (FileXLInvalid=Yes, IsPattern=Yes, EndRuleToken=Yes)
    TKG_IF = IF:[^\w\d] (IsPattern=Yes)
    TKG_THEN = THEN:[^\w\d] (IsPattern=Yes, EndRuleToken=Yes)
    TKG_BLOCK_ELSEIF = ELSIF:[^\w\d] (IsPattern=Yes)
    TKG_ELSE_AND_DEFAULT = ELSE:[^\w\d] (IsPattern=Yes, EndRuleToken=Yes)
    TKG_BLOCK_ENDIF = END_IF:[^\w\d] (IsPattern=Yes, EndRuleToken=Yes)
    TKG_SWITCH = CASE:[^\w\d] (IsPattern=Yes, FileXLInvalid=Yes)
    TKG_ENDSWITCH_NOBREAK = END_CASE:[^\w\d] (FileXLInvalid=Yes, IsPattern=Yes, EndRuleToken=Yes)
    TKG_WHILE = WHILE:[^\w\d] (FileXLInvalid=Yes, IsPattern=Yes)
    TKG_ENDWHILE = END_WHILE:[^\w\d] (FileXLInvalid=Yes, IsPattern=Yes, EndRuleToken=Yes)
    TKG_DO = REPEAT:[^\w\d] (FileXLInvalid=Yes, IsPattern=Yes, EndRuleToken=Yes)
    TKG_ENDDO_UNTIL = UNTIL:[^\w\d] (FileXLInvalid=Yes, IsPattern=Yes)
    TKG_ENDDO_POSTCOND = END_REPEAT:[^\w\d] (FileXLInvalid=Yes, IsPattern=Yes, EndRuleToken=Yes)
    TKG_BREAK = EXIT:[^\w\d] (FileXLInvalid=Yes, IsPattern=Yes)
    TKG_RETURN = RETURN:[^\w\d] (FileXLInvalid=Yes, IsPattern=Yes)
    TKG_IEC_SEL_FN = SEL:[^\w\d] (FileXLInvalid=Yes, IsPattern=Yes)
    TKG_IEC_MUX_FN = MUX:[^\w\d] (FileXLInvalid=Yes, IsPattern=Yes)
    TKG_TIME_LITERAL = time#\-[dDhHmMsS_\.\d]+|time#[dDhHmMsS_\.\d]+|t#\-[dDhHmMsS_\.\d]+|t#[dDhHmMsS_\.\d]+ (CaseSensitive=no, IsPattern=yes)
    TKG_DATE_AND_TIME_LITERAL = DT#[12]\d\d\d\-[\d\:\-]*|DATE_AND_TIME#[12]\d\d\d\-[\d\:\-]* (CaseSensitive=no, IsPattern=yes)
    TKG_DATE_LITERAL = D#[12]\d\d\d\-[\d\-]*|DATE#[12]\d\d\d\-[\d\-]* (CaseSensitive=no, IsPattern=yes)
    TKG_TIME_OF_DAY_LITERAL = TOD#\d[\d\:\.]*|TIME_OF_DAY#\d[\d\:\.]* (CaseSensitive=no, IsPattern=yes)
    TKG_ASSIGN_EQ = :=
    TKG_OPEN_IP_EXTENSION = {
    TKG_CLOSE_IP_EXTENSION = }
    TKG_IEC_OPEN_TYPE = TYPE:[^\w\d] (IsPattern=Yes)
    TKG_IEC_CLOSE_TYPE = END_TYPE:[^\w\d] (IsPattern=Yes, EndRuleToken=Yes)
    TKG_VAR = VAR:[^\w\d] (IsPattern=Yes)
    TKG_VAR_GLOBAL = VAR_GLOBAL:[^\w\d] (IsPattern=Yes)
    TKG_VAR_INPUT = VAR_INPUT:[^\w\d] (IsPattern=Yes)
    TKG_VAR_OUTPUT = VAR_OUTPUT:[^\w\d] (IsPattern=Yes)
    TKG_VAR_IN_OUT = VAR_IN_OUT:[^\w\d] (IsPattern=Yes)
    TKG_VAR_END = END_VAR:[^\w\d] (IsPattern=Yes, EndRuleToken=Yes)
    TKG_VAR_RETAIN = RETAIN:[^\d\w] (IsPattern=Yes)
    TKG_IP_RETAIN = IP_RETAIN:[^\d\w] (IsPattern=Yes)
    TKG_AT = AT:[^\d\w] (IsPattern=Yes)
    TKG_PLC = PLC:[^\d\w] (IsPattern=Yes)
    TKG_PV_UNDECL = UNRETAIN_VAR:[^\d\w] (IsPattern=Yes)
    TKG_VARSYNCH_IP = IP_SYNCH:[^\d\w] (IsPattern=Yes)
    TKG_VARSYNCH_PATH = PATH_SYNCH:[^\d\w] (IsPattern=Yes)
    TKG_CONSTANT = CONSTANT:[^\d\w] (IsPattern=Yes)
    TKG_VARSCOPE_IP_GLOBAL = IP_GLOBAL:[^\w\d] (IsPattern=Yes)
    TKG_VARSCOPE_SHARED_IP_GLOBAL = SHARED_IP_GLOBAL:[^\w\d] (IsPattern=Yes)
    TKG_VARSCOPE_NC_GLOBAL = NC_GLOBAL:[^\w\d] (IsPattern=Yes)
    TKG_VARSCOPE_PLC_GLOBAL = PLC_GLOBAL:[^\w\d] (IsPattern=Yes)
    TKG_VARSCOPE_IP_LOCAL = LOCAL:[^\w\d] (IsPattern=Yes)
    TKG_IEC_NAMESPACE_SPEC = :: (IsPattern=No)
    TKG_IEC_DATATYPE_SPEC = : (IsPattern=No)
    TKG_IEC_ARRAY = ARRAY:[^\w\d] (IsPattern=Yes)
    TKG_IEC_OF = OF:[^\w\d] (IsPattern=Yes)
    TKG_IEC_DELIM = ; (EndRuleToken=Yes)
    TKG_IEC_OPEN_STRUCT = STRUCT:[^\w\d] (IsPattern=Yes)
    TKG_IEC_CLOSE_STRUCT = END_STRUCT:[^\w\d] (IsPattern=Yes)
    TKG_BITWISE_LP_BINARY_AND = AND:[^\w\d] (IsPattern=Yes)
    TKG_BITWISE_LP_BINARY_OR = OR:[^\w\d] (IsPattern=Yes)
    TKG_BITWISE_LP_BINARY_XOR = XOR:[^\w\d] (IsPattern=Yes)
    TKG_BITWISE_UNARY_COMPLEMENT = NOT:[^\w\d] (IsPattern=Yes)
    TKG_COMP_EXACT_BINARY_GREATER_THAN_OR_EQ = >=
    TKG_COMP_EXACT_BINARY_LESS_THAN_OR_EQ = <=
    TKG_COMP_EXACT_BINARY_EQUAL_TO = =
    TKG_COMP_EXACT_BINARY_NOT_EQUAL_TO = <>
    TKG_COMP_EXACT_BINARY_GREATER_THAN = >
    TKG_COMP_EXACT_BINARY_LESS_THAN = <
    TKG_ARITH_BINARY_PLUS = +
    TKG_ARITH_BINARY_MINUS = -
    TKG_ARITH_BINARY_POWER = **
    TKG_ARITH_BINARY_MULTIPLY = *
    TKG_ARITH_BINARY_DIVIDE = /
    TKG_ARITH_BINARY_MODULO = MOD:[^\w\d] (IsPattern=Yes)
    TKG_PRAGMA = #pragma:[^\w\d] (IsPattern=Yes, FollowedBy=TKG_IDENTIFIER)
    TKG_INCLUDE = #include:[^\w\d] (IsPattern=Yes)
    TKG_PROG_START = PROGRAM:[^\w\d] (IsPattern=Yes, FollowedBy=TKG_PROG_NAME)
    TKG_PROG_NAME = _INIT:[^\w\d]|_CYCLIC:[^\w\d]|_EXIT:[^\w\d]|_MAIN:[^\w\d] (IsPattern=Yes, EndRuleToken=Yes)
    TKG_PROG_END = END_PROGRAM:[^\w\d] (IsPattern=Yes, EndRuleToken=Yes)
    TKG_SUBPROG_START = FUNCTION:[^\w\d] (IsPattern=Yes)
    TKG_SUBPROG_END = END_FUNCTION:[^\w\d] (IsPattern=Yes, EndRuleToken=Yes)
    TKG_FUB_DECL = FUNCTION_BLOCK:[^\w\d] (IsPattern=Yes)
    TKG_FUB_END = END_FUNCTION_BLOCK:[^\w\d] (IsPattern=Yes, EndRuleToken=Yes)
    TKG_RETURN = RETURN:[^\w\d] (IsPattern=Yes)
    TKG_ACCESS = ACCESS:[^\w\d] (IsPattern=Yes)
    TKG_DEREF_OP = ^
    TKG_ACTION = ACTION:[^\w\d] (IsPattern=Yes)
    TKG_ACTION_END = END_ACTION:[^\w\d] (IsPattern=Yes, EndRuleToken=Yes)
    TKG_IEC_TYPED_VALUE = \w#:[\w\d\+\-]|\w[\w\d]+#:[\w\d\+\-] (IsPattern=Yes)
    TKG_PARAM_PREFIX = $R:[^\w\d]|$P:[^\w\d]|$MW:[^\w\d]|$ML:[^\w\d]|$MF:[^\w\d]|$EXW:[^\w\d]|$EXL:[^\w\d]|$EXF:[^\w\d]|$EXB:[^\w\d] (IsPattern=Yes)
    TKG_IDENTIFIER = \w|\w[\w\d$]+|$[\w\d$]+ (IsPattern=Yes)
    TKG_INIT_IDENTIFIER = \w|\w[\w\d$]+|$[\w\d$]+ (IsPattern=Yes, Disabled=Yes)
  StringChars (AsciiStringStart=', AsciiStringEnd=', UTF16StringStart=", UTF16StringEnd=")
    EscapeSeq (Search=$N, CaseSensitive=Yes, ReplaceValue=10)
    EscapeSeq (Search=$n, CaseSensitive=Yes, ReplaceValue=10)
    EscapeSeq (Search=$L, CaseSensitive=Yes, ReplaceValue=10)
    EscapeSeq (Search=$l, CaseSensitive=Yes, ReplaceValue=10)
    EscapeSeq (Search=$P, CaseSensitive=Yes, ReplaceValue=12)
    EscapeSeq (Search=$p, CaseSensitive=Yes, ReplaceValue=12)
    EscapeSeq (Search=$R, CaseSensitive=Yes, ReplaceValue=13)
    EscapeSeq (Search=$r, CaseSensitive=Yes, ReplaceValue=13)
    EscapeSeq (Search=$T, CaseSensitive=Yes, ReplaceValue=9)
    EscapeSeq (Search=$t, CaseSensitive=Yes, ReplaceValue=9)
    EscapeSeq (Search=$', CaseSensitive=Yes, ReplaceStr=')
    EscapeSeq (Search=$", CaseSensitive=Yes, ReplaceStr=")
    EscapeSeq (Search=$[\dA-Fa-f]+, IsPattern=Yes, CaseSensitive=Yes, ReplaceEncodingBase=16)
    EscapeSeq (Search=$$, ReplaceStr=$)
    EscapeSeq (Search=$, ReplaceStr=)
```

- Data object Logical/GmcIpConfig/gmciplog (Cnc, version 3.14.3) (no source held here)

- Data object Logical/GmcIpConfig/gmcipmxd (Cnc, version 3.14.3) (no source held here)

- Data object Logical/GmcIpUserConfig/gmcipubr (Cnc, version 3.14.3) (no source held here)

- Data object Logical/GmcIpUserConfig/gmcipuc (Cnc, version 3.14.3) (no source held here)

- Data object Logical/GmcIpUserConfig/gmcipui (Cnc, version 3.14.3) (no source held here)

- Data object Logical/GmcIpUserConfig/gmcipus (Cnc, version 3.14.3) (no source held here)

- Data object Logical/GmcIpUserConfig/gmcipusm (Cnc, version 3.14.3) (no source held here)

- Data object Logical/GmcIpUserConfig/gmcipvar (Cnc, version 3.14.3) (no source held here)

### AS3500_Par.typ - not listed in the package file held
```iecst
TYPE
	AS3500HS_Control_Rec_typ : 	STRUCT
		N_Targets_On_Dial : UDINT;
		Enable_Cure : ARRAY[0..1]OF UDINT;
	END_STRUCT;
	AS3500HS_Control_Cfg_typ : 	STRUCT
		N_Encoder_Bits_SingleTurn : UDINT;
		Encoder_Position_Home : UDINT;
		Debounce_PiP : Debounce_Config_Struct;
		Threshold_AccelDecel_Trans_RPM : REAL;
		T_Exit_Decel_Automatically : REAL;
		Sim_Encoder : UDINT;
		Sim_Encoder_Cycles : UDINT;
		Sim_Encoder_Counts : UDINT;
		Target_Present_Pulse_Time_S : REAL;
	END_STRUCT;
END_TYPE
```

### Enumerations.typ - not listed in the package file held
```iecst
TYPE
	CMA_Arimat_PrcsState_Enum :
		(
		PRCS_STATE_INIT,
		PRCS_STATE_IDLE,
		PRCS_STATE_WAIT_LOADER,
		PRCS_STATE_FEED_OFFSET,
		PRCS_STATE_BLADE_CREASER,
		PROCESS_STATE_FINISHING,
		PROCESS_STATE_ERROR
		);
	CMA_Arimat_MachineState_Enum :
		(
		MACHINE_STATE_INIT,
		MACHINE_STATE_IDLE,
		MACHINE_STATE_RUNNING,
		MACHINE_STATE_ERRORSTOP,
		MACHINE_STATE_MANUAL_CTRL
		);
END_TYPE
```

### IO.typ - not listed in the package file held
```iecst
TYPE
	IO_Status_typ : 	STRUCT
		iEmergencyStop : BOOL;
		oFolderInsertOK : BOOL;
		iProductInPlace : BOOL;
		oWarningLight : BOOL;
	END_STRUCT;
	IO_Motor_typ : 	STRUCT
		iMotorTemperatureSwitch : BOOL;
		iBladeEngineStopSensor : BOOL;
		oCreasingEngineClutch : BOOL;
	END_STRUCT;
	CMA_Arimat_IO_typ : 	STRUCT
		Status : IO_Status_typ;
		Motor : IO_Motor_typ;
	END_STRUCT;
END_TYPE
```

### RecipeConfig.typ - not listed in the package file held
```iecst
TYPE
	Global_Rec_typ : 	STRUCT
		MagicPrefix : UDINT;
		New_Member : USINT;
		MagicSuffix : UDINT;
	END_STRUCT;
	Global_Cfg_typ : 	STRUCT
		MagicPrefix : UDINT;
		New_Member : USINT;
		MagicSuffix : UDINT;
	END_STRUCT;
END_TYPE
```

### GlobalConstants.var - not listed in the package file held
```iecst
VAR CONSTANT
	FORCEIO_ACCESS_LEVEL : UINT := 1;
	CONFIG_ACCESS_LEVEL : UINT := 2;
	RECIPE_ACCESS_LEVEL : UINT := 1;
	DEFINE_MENU_L_HIDE_TIMEOUT_MS : UDINT := 7000;
	DEFINE_MENU_R_HIDE_TIMEOUT_MS : UDINT := 7000;
	DEFINE_HMI_SPLASHSCREEN_TO_MS : UDINT := 5000;
	MAX_IDX_VALVES : USINT := 1;
	MAX_IDX_TARGETS : UDINT := 50; (*Total number of VBlocks that may EVER be installed on the system.  *)
	MAX_RPM_GAUGE : REAL := 25;
	COLORBAR_FLASH_TO : TIME := T#750ms;
	MAX_IDX_TOTAL_RECIPES : UINT := 100;
	DEFINE_LOGIN_TO : REAL := 600; (*// at timer DEFINE_LOGIN_TO * 1000 *60*)
	DEFINE_TN_VELCALC : REAL := 0.1;
END_VAR
```

### varPkg.var - not listed in the package file held
```iecst
(*IO Values*)
VAR
	IO : CMA_Arimat_IO_typ;
END_VAR
(*<--------------------------------------------->*)
(*Control State Machine States*)
VAR
	MachineState : CMA_Arimat_MachineState_Enum;
	ProcessState : CMA_Arimat_PrcsState_Enum;
END_VAR
(*<--------------------------------------------->*)
(*<--------------------------------------------->*)
(**)
(*<--------------------------------------------->*)
(*<--------------------------------------------->*)
(**)
(*<--------------------------------------------->*)
(*Insert your comment here.*)
(*Insert your comment here.*)
(*Insert your comment here.*)
(*Insert your comment here.*)
```

### AlarmsWarnings.typ
```iecst
TYPE
	HERNON_Alarm_Dispense_typ : 	STRUCT
		Valve_Not_Ready : BOOL;
		Valve_Ready_Neg_Edge_Error : BOOL;
		EdgeGenError : BOOL;
		Max_Time_Fractional_Offset : BOOL;
	END_STRUCT;
END_TYPE
```

### Program Logical/Application/Dispense/Valves

#### Variables.var
```iecst
VAR
	Debug_Stats_LastCycle : AS3500_Disp_Debug_typ;
	ii_valves : UDINT := 0;
	ValveReadyFailCount : {REDUND_UNREPLICABLE} DINT;
	ValveReadyFailCount_LastCycle : {REDUND_UNREPLICABLE} DINT;
	CycleCount : {REDUND_UNREPLICABLE} DINT;
	CycleCount_LastCycle : {REDUND_UNREPLICABLE} DINT;
END_VAR
```

#### Main.st
```iecst
PROGRAM _INIT

	//Valve names for alarm groups-
	ValveFBK[0].Name := 'Valve 1';
	ValveFBK[1].Name := 'Valve 2';

END_PROGRAM

PROGRAM _CYCLIC
	FOR ii_valves :=0 TO MAX_IDX_VALVES BY 1 DO

		IF gRecCfg.active.Cfg.Dispense[ii_valves].Disable = 1 THEN
			gRecCfg.active.Rec.Dispense[ii_valves].Enable := FALSE;
		END_IF;

		ValveFBK[ii_valves].pCounterValveNotRdy := ADR(gStatistics.Debug.Valve_Not_Rdy[ii_valves].Count);
		ValveFBK[ii_valves].pCyclesCounter := ADR(gStatistics.Debug.Disp_Cycle_Count[ii_valves].Count);
		ValveFBK[ii_valves].iVBlockFractionalPosition := Position.Target_Fractional_Position_Pct;
		ValveFBK[ii_valves].iX2XNettime := ControlIO.iX2XNettime;
		ValveFBK[ii_valves].Recipe := ADR(gRecCfg.active.Rec.Dispense[ii_valves]);
		ValveFBK[ii_valves].Config := ADR(gRecCfg.active.Cfg.Dispense[ii_valves]);
		ValveFBK[ii_valves].IO := ADR(ValveIO[ii_valves]);
		ValveFBK[ii_valves].Alarms := ADR(gAlarms.Sureshot3500[ii_valves]);
		ValveFBK[ii_valves]();

		IF gStatistics.Debug.Valve_Not_Rdy[ii_valves].Count > Debug_Stats_LastCycle.Valve_Not_Rdy[ii_valves].Count THEN
			gStatistics.Debug.Valve_Not_Rdy[ii_valves].Latch_Position := Position;
		END_IF;

	END_FOR;

	Debug_Stats_LastCycle := gStatistics.Debug;

END_PROGRAM

PROGRAM _EXIT
	(* Insert code here *)

END_PROGRAM

//Notes-
//-Four valves were included such that they could be substituted.  Can be disabled if functionality is undesirable.
```

### Program Logical/Application/Master/ControlLogic

#### Variables.var
```iecst
VAR
	Dashboard_Hide_Encoder_Sim : USINT;
	ii_valves : USINT;
	CMD_Set_Home_Pos_0 : BOOL;
	CMD_Set_Current_Pos_As_Home : BOOL;
	CMD_Reset_Statistics : BOOL;
	encoder_diff_counts : INT;
	Multiturn_Absolute_Position : DINT;
	PositionValue : UINT;
	ShiftBits : UINT;
	Timer_Total_Runtime : TON;
	Timer_Pulse_Target_Present : TON;
	STATUS_LIGHT_FLASH : FLASH;
	Flag_Cure_Error_Exists : BOOL;
	Flag_Valve_Error_Exists : BOOL;
END_VAR
```

#### Action_Manage_Update_Total_Runtime.st
```iecst
ACTION Action_Manage_Update_Total_Runtime:

	IF bgTimerIsTimeOut(Timer_Total_Runtime) THEN
		gStatistics.total_runtime := gStatistics.total_runtime + 1;
		bgTimerStart(Timer_Total_Runtime, 1000);

		gStatistics.runtime_h := gStatistics.total_runtime / 3600;
		gStatistics.runtime_m := (gStatistics.total_runtime/60) MOD 60;
		gStatistics.runtime_s := gStatistics.total_runtime MOD 60;
	END_IF;

	bgTimerCyclic(Timer_Total_Runtime);

END_ACTION
```

#### Action_Set_Colorbar_IO.st
```iecst
ACTION Action_Set_Colorbar_IO:

	CASE ColorBar OF
		COLOR_NONE:
			StatusIO.oStatusColor.Red := FALSE;
			StatusIO.oStatusColor.Green := FALSE;
			StatusIO.oStatusColor.Blue := FALSE;

		COLOR_GREEN_FLASH:
			StatusIO.oStatusColor.Red := FALSE;
			StatusIO.oStatusColor.Green := STATUS_LIGHT_FLASH.bFlashOut;
			StatusIO.oStatusColor.Blue := FALSE;

		COLOR_GREEN:
			StatusIO.oStatusColor.Red := FALSE;
			StatusIO.oStatusColor.Green := TRUE;
			StatusIO.oStatusColor.Blue := FALSE;

		COLOR_GREEN_BLUE_ALTERNATE:
			StatusIO.oStatusColor.Red := FALSE;
			StatusIO.oStatusColor.Green := STATUS_LIGHT_FLASH.bFlashOut;
			StatusIO.oStatusColor.Blue := NOT STATUS_LIGHT_FLASH.bFlashOut;

		COLOR_RED:
			StatusIO.oStatusColor.Red := TRUE;
			StatusIO.oStatusColor.Green := FALSE;
			StatusIO.oStatusColor.Blue := FALSE;

		COLOR_GREEN_RED_ALTERNATE:
			StatusIO.oStatusColor.Red := STATUS_LIGHT_FLASH.bFlashOut;
			StatusIO.oStatusColor.Green := NOT STATUS_LIGHT_FLASH.bFlashOut;
			StatusIO.oStatusColor.Blue := FALSE;

	END_CASE;

	STATUS_LIGHT_FLASH(TimeOn := COLORBAR_FLASH_TO, TimeOff := COLORBAR_FLASH_TO);

END_ACTION
```

#### Main.st
```iecst
PROGRAM _INIT
	VelCalc_DT_Element.Enable := 1;
	VelCalc_DT_Element.Gain := 1;
	VelCalc_DT_Element.TimeConstant := DEFINE_TN_VELCALC;
	VelCalc_DT_Element();

	gState := STATE_INIT;
END_PROGRAM

PROGRAM _CYCLIC

	//Action for testing the PiP sensor->
	Action_Test_PiP_Trigger;

//	ControlIO.Inspection.oInspectionGood := ValveIO[0].oDispTrigger;
	//	ControlIO.Inspection.oInspectionValid := ValveIO[1].oDispTrigger;

	//Have to check for the following...
	IF gRecCfg.active.Cfg.Control.N_Encoder_Bits_SingleTurn = 0 OR gRecCfg.active.Rec.Control.N_Targets_On_Dial = 0 THEN
		gAlarms.Control.Invalid_Par := TRUE;
		RETURN; //...Otherwise machine will go into service mode due to integer div. 0 error
	END_IF;

	//Handle commands from HMI (Home pos., reset stats)
	Action_HMI_Commands_Handler;
	//Calc current pos/vel of the dial for triggering purposes-
	Action_Dial_Position_Velocity_Calc;

	IF gState <> STATE_ERROR AND (NOT (StatusIO.iProcessStopRelay[0] AND StatusIO.iProcessStopRelay[1])) THEN
		gState := STATE_ERROR;
	END_IF;

	//Manage PiP target sensor debounce to prevent "dirty edge" switching->
	ControlIO.PiP_Sensor_Debounce.pConfigVals := ADR(gRecCfg.active.Cfg.Control.Debounce_PiP);
	ControlIO.PiP_Sensor_Debounce(input := ControlIO.iTargetPiP);

	//On target index, reset "TargetInfoArray" index for the target that has just moved in front of the PiP sensor (all values to 0)
	IF Position.Current_Target <> Position_LastCycle.Current_Target THEN
		brsmemset(ADR(TargetInfoArray[Position.Current_Target]), 0, SIZEOF(Target_typ));
	END_IF;

	//On + edge of SW debounced PiP sensor, enter info. into array-
	IF ControlIO.PiP_Sensor_Debounce.Signal_Debounced = 1 AND ControlIO_LastCycle.PiP_Sensor_Debounce.Signal_Debounced = 0 THEN
		IF TargetInfoArray[Position.Current_Target].VBlock_Occupied THEN //Handler for diagnostics purposes when there are 2 + edges on the same target
			gStatistics.Count_PiP_Twice_Single_Targ.Count := gStatistics.Count_PiP_Twice_Single_Targ.Count + 1;
			gStatistics.Count_PiP_Twice_Single_Targ.Latch_Position := Position;
		ELSE
			gStatistics.VBlock_Fraction_Pos_Last_Edge := Position.Target_Fractional_Position_Pct;
			TargetInfoArray[Position.Current_Target].VBlock_Occupied := TRUE;
			gStatistics.Total_Num_Targets := gStatistics.Total_Num_Targets + 1;
			bgTimerStart(Timer_Pulse_Target_Present, Tms(gRecCfg.active.Cfg.Control.Target_Present_Pulse_Time_S));
		END_IF;
	END_IF;

	ControlIO.oTargetPresent := NOT bgTimerIsTimeOut(Timer_Pulse_Target_Present);

	Flag_Cure_Error_Exists := FALSE;

	IF gRecCfg.active.Rec.Control.Enable_Cure[0] = 1 AND NOT CureIO.iUVCuringChannelOK[0] THEN
		Flag_Cure_Error_Exists := TRUE;
	END_IF;

	IF gRecCfg.active.Rec.Control.Enable_Cure[1] = 1 AND NOT CureIO.iUVCuringChannelOK[1] THEN
		Flag_Cure_Error_Exists := TRUE;
	END_IF;

	//Flag for valve error, reset on every cycle->
	Flag_Valve_Error_Exists := FALSE;

	FOR ii_valves := 0 TO MAX_IDX_VALVES BY 1 DO
		//Set values of current target index in front of each dispense unit
		Control.Dispense[ii_valves].Current_Target_At_Dispense_Unit := ((Position.Current_Target) + (gRecCfg.active.Rec.Control.N_Targets_On_Dial - gRecCfg.active.Rec.Dispense[ii_valves].Target_Offset)) MOD (gRecCfg.active.Rec.Control.N_Targets_On_Dial);
		Control.Dispense[ii_valves].Target_Fractional_Position_Pct := Position.Target_Fractional_Position_Pct;

		IF ValveFBK[ii_valves].oState = DISPENSE_STATE_ERROR THEN
			Flag_Valve_Error_Exists := TRUE;
		END_IF;

		gStatistics.Dispense_Discrepancy := UDINT_TO_DINT(gStatistics.Debug.Disp_Trigger_Count[ii_valves].Count - gStatistics.Debug.Disp_Cycle_Count[ii_valves].Count);
	END_FOR;

	CASE gState OF
		STATE_INIT:
			ColorBar := COLOR_NONE;
			StatusIO.oSystemNeedsAttention := FALSE;
			StatusIO.oRunningReady := FALSE;

			CureIO.oUVCureChannel[0] := FALSE;
			CureIO.oUVCureChannel[1] := FALSE;

			gState := STATE_IDLE;
		STATE_IDLE:
			ColorBar := COLOR_GREEN_FLASH;
			StatusIO.oSystemNeedsAttention := FALSE;
			StatusIO.oRunningReady := TRUE;

			CureIO.oUVCureChannel[0] := gRecCfg.active.Rec.Control.Enable_Cure[0] = 1;
			CureIO.oUVCureChannel[1] := gRecCfg.active.Rec.Control.Enable_Cure[1] = 1;

			IF Flag_Valve_Error_Exists OR Flag_Cure_Error_Exists THEN
				gState := STATE_ERROR;
			ELSIF ControlIO.iRunCmd THEN
				gState := STATE_RUNNING;
			END_IF;

		STATE_RUNNING:
			ColorBar := COLOR_GREEN;
			Action_Dispense_TriggerFinger;
			StatusIO.oSystemNeedsAttention := FALSE;
			StatusIO.oRunningReady := TRUE;

			CureIO.oUVCureChannel[0] := gRecCfg.active.Rec.Control.Enable_Cure[0] = 1;
			CureIO.oUVCureChannel[1] := gRecCfg.active.Rec.Control.Enable_Cure[1] = 1;

			Action_Manage_Update_Total_Runtime;

			IF NOT ControlIO.iRunCmd THEN
				gState := STATE_IDLE;
			ELSIF Flag_Valve_Error_Exists OR Flag_Cure_Error_Exists THEN
				gState := STATE_ERROR;
			END_IF;

		STATE_ERROR:
			ColorBar := COLOR_RED;
			StatusIO.oSystemNeedsAttention := TRUE;
			StatusIO.oRunningReady := FALSE;

			CureIO.oUVCureChannel[0] := FALSE;
			CureIO.oUVCureChannel[1] := FALSE;

			IF StatusIO.iProcessStopRelay[0] AND StatusIO.iProcessStopRelay[1] AND (StatusIO.iClearError AND NOT StatusIO_LastCycle.iClearError) (*AND (NOT Flag_Valve_Error_Exists)*) AND (NOT Flag_Cure_Error_Exists) THEN
				FOR ii_valves := 0 TO MAX_IDX_VALVES BY 1 DO
					ValveFBK[ii_valves].iReset := TRUE;
				END_FOR;

				gState := STATE_IDLE;
			END_IF;

	END_CASE;

	bgTimerCyclic(Timer_Pulse_Target_Present);

	Action_Set_Colorbar_IO;

	Position_LastCycle := Position;
	Position_SHL_LastCycle := Position_SHL;

	CureIO_LastCycle := CureIO;
	StatusIO_LastCycle := StatusIO;
	ControlIO_LastCycle := ControlIO;
END_PROGRAM

PROGRAM _EXIT

END_PROGRAM
```

### USB_Mount_types.typ
```iecst
TYPE
	USB_Global_SM_Enum :
		(
		STEP_GET_NODE_LIST := 0,
		STEP_READ_DEVICE_DATA := 1,
		STEP_USB_ERROR := 2,
		STEP_CHECK_MOUNT_STATUS := 3,
		STEP_MOUNT_DISMOUNT := 4,
		STEP_WAIT_NODE_RESCAN := 5
		);
	Dev_Mount_Statuses :
		(
		DEVICE_NOT_CONNECTED := 0,
		DEVICE_NOT_MOUNTED := 1,
		DEVICE_MOUNTING := 2,
		DEVICE_MOUNTED := 3,
		DEVICE_DISCON_WHILE_MOUNTED := 4,
		DEVICE_UNMOUNTING := 5,
		DEVICE_UNMOUNTED_CONNECTED := 6,
		DEVICE_NOT_MOUNTABLE := 7,
		DEVICE_DISMOUNT_ERROR := 8,
		DEVICE_MOUNT_ERROR := 9,
		DEVICE_IS_TECHGUARD_DONGLE := 10
		);
	USB_FBK_typ : 	STRUCT
		Link_Device : DevLink;
		Unlink_Device : DevUnlink;
	END_STRUCT;
	USB_Data_typ : 	STRUCT
		usb_node_info_connected : usbNode_typ;
		usb_node_info_to_connect : usbNode_typ;
		device_descriptor : usbDeviceDescr_typ;
		device_param : STRING[80];
		device_name : STRING[80];
	END_STRUCT;
	USB_Object_typ : 	STRUCT
		FBK : USB_FBK_typ;
		Data : USB_Data_typ;
		Err : BOOL;
		Force_Dismount : BOOL;
		Status : Dev_Mount_Statuses;
		Mounted : BOOL;
	END_STRUCT;
END_TYPE
```

### Program Logical/Auxiliary_Services_Control/Recipe_Handling
